(* IEC 61131-3 sources: Industry-PLC-LLM/data/PLCBEAD_repo/PLCBEAD_PLCEmbed-main/PLC-BEAD/Source/OpenPLCv2 (part 10) *)

(* ---- TN_SEND_ROWS.ST ---- *)
TYPE
  oscat_IP_FIFO128_DATA  : ARRAY [1..128] OF BYTE;
  oscat_Mailbox  : ARRAY [1..16] OF BYTE;

  oscat_IP_FIFO_DATA :
  STRUCT
    X       : oscat_IP_FIFO128_DATA; (* IP_ID FIFO Speicher          *)
    Y       : oscat_IP_FIFO128_DATA; (* IP_ID Z�hler                 *)
    ID      : BYTE;                  (* h�chste vergabene id         *)
    MAX_ID  : BYTE;                  (* maximal Anmeldungen pro ID   *)
    INIT    : BOOL;                  (* Initialisierung durchgef�hrt *)
    EMPTY   : BOOL;                  (* FIFO leer                    *)
    FULL    : BOOL;                  (* FIFO voll                    *)
    TOP     : INT;                   (* maximale anzahl in FIFO      *)
    NW      : INT;                   (* Schreibzeiger                *)
    NR      : INT;                   (* Lesezeiger                   *)
  END_STRUCT;

  oscat_IP_C:
  STRUCT
    C_MODE:			BYTE;          		(*W Mode: TCP/UCP AKTIV/PASSIV                               *)
    C_PORT:         WORD;          		(*W Portnummer                                               *)
    C_IP:           DWORD;         		(*W IP-Adresse gepackt wwxxyyzz = www.xxx.yyy.zzz            *)
    C_STATE:        BYTE;          		(*R Verbindungsstatus ON/OFF + Flanke ON/OFF                 *)
    C_ENABLE:       BOOL;          		(*W Freigabe f�r Connect                                     *)
    R_OBSERVE:      BOOL;          		(*W Empfang ueberwachen                                      *)
    TIME_RESET:     BOOL;          		(*W Alle Timer ruecksetzen                                   *)
    ERROR:          DWORD;         		(*R vvwwxxyy (vv = CON_ERROR, ww = SEN_ERROR, xx = REC_ERROR *)
    FIFO:           oscat_IP_FIFO_DATA; (*I IP FIFO Struktur                                         *)
    MAILBOX:		oscat_Mailbox;		(*I Mailbox: Datenbereich f�r Bausteindatenaustausch         *)
    END_STRUCT;
END_TYPE

TYPE

  oscat_NW_BUF_LONG  : ARRAY [0..4095] OF BYTE;

  oscat_NETWORK_BUFFER :
  STRUCT
    SIZE   : UINT;
    BUFFER : oscat_NW_BUF_LONG;
  END_STRUCT;

END_TYPE

TYPE

  bya_TN_CHAR:       	ARRAY [0..1919] OF BYTE;
  bya_TN_BACKUP:     	ARRAY [0..1919] OF BYTE;
  bya_TN_COLOR:      	ARRAY [0..1919] OF BYTE;
  bya_TN_Line_Update:	ARRAY [0..23]   OF BOOL;

  us_TN_SCREEN :
  STRUCT
    bya_CHAR:			bya_TN_CHAR;
    bya_COLOR:			bya_TN_COLOR;
    bya_BACKUP:			bya_TN_BACKUP;
    bya_Line_Update:	bya_TN_Line_Update;

    by_Input_Exten_Code:    BYTE;
    by_Input_ASCII_Code:    BYTE;
    bo_Input_ASCII_IsNum:   BOOL;
    in_Page_Number:        	INT;                (* aktive Seiten-Nr.              *)
    in_Cursor_X:           	INT;                (* Cursor X-Position              *)
    in_Cursor_Y:           	INT;                (* Cursor Y-Position              *)
    in_EOS_Offset:         	INT;                (* End of String Offset           *)
    by_Clear_Screen_Attr:  	BYTE;               (* Clear-Screen Attr              *)
    bo_Clear_Screen:       	BOOL;               (* Clear-Screen ausl�sen          *)
    bo_Modal_Dialog:       	BOOL;               (* Modaler Dialog ist aktiv       *)
    bo_Menue_Bar_Dialog:   	BOOL;               (* Menue Dialog ist aktiv         *)

  END_STRUCT;
END_TYPE

FUNCTION INT_TO_BCDC:BYTE

	VAR_INPUT
		IN :	INT;
	END_VAR

	INT_TO_BCDC := SHL(INT_TO_BYTE(IN / INT#10),4) OR INT_TO_BYTE(in MOD INT#10);

END_FUNCTION

FUNCTION_BLOCK TN_SEND_ROWS_Block

  VAR_IN_OUT
    IP_C :	oscat_IP_C;
    S_BUF :	oscat_NETWORK_BUFFER;
    Xus_TN_SCREEN :	us_TN_SCREEN;
  END_VAR

  VAR_INPUT
    S_BUF_SIZE :	INT;
  END_VAR

  VAR
    in_Line_Count :	INT;
    in_Col_Count :	INT;
    in_Last_Row_Index :	INT;
    bo_Break_Loop :	BOOL;
    in_Row_Count :	INT;
    in_Offset :	INT;
    in_Write_Index :	INT;
    in_Write_Index_Backup :	INT;
    by_Cur_Color :	BYTE;
    by_last_Color :	BYTE;
    in_Write_Stop :	INT;
  END_VAR

  IF (IP_C.C_STATE < BYTE#127 OR S_BUF.SIZE > UINT#0) THEN
    RETURN;
  END_IF;

  in_Write_Index := UINT_TO_INT(S_BUF.SIZE) - 1;

  in_Write_Index_Backup := in_Write_Index;

  IF (IP_C.C_STATE = BYTE#254) OR (Xus_TN_SCREEN.bo_Clear_Screen) THEN

    Xus_TN_SCREEN.bo_Clear_Screen := FALSE;

    FOR in_Line_Count := INT#00 TO INT#23 DO
      Xus_TN_SCREEN.bya_Line_Update[in_Line_Count] := TRUE;
    END_FOR;

    in_Write_Index := in_Write_Index + INT#1;
    S_BUF.BUFFER[in_Write_Index] := BYTE#16#1B;
    in_Write_Index := in_Write_Index + INT#1;
    S_BUF.BUFFER[in_Write_Index] := BYTE#16#5B;
    in_Write_Index := in_Write_Index + INT#1;
    S_BUF.BUFFER[in_Write_Index] := BYTE#16#30;
    in_Write_Index := in_Write_Index + INT#1;
    S_BUF.BUFFER[in_Write_Index] := BYTE#16#3B;
    in_Write_Index := in_Write_Index + INT#1;
    S_BUF.BUFFER[in_Write_Index] := BYTE#16#33;

    in_Write_Index := in_Write_Index + INT#1;
    S_BUF.BUFFER[in_Write_Index] := (SHR(Xus_TN_SCREEN.by_Clear_Screen_Attr,4) OR BYTE#16#30);

    in_Write_Index := in_Write_Index + INT#1;
    S_BUF.BUFFER[in_Write_Index] := BYTE#16#3B;
    in_Write_Index := in_Write_Index + INT#1;
    S_BUF.BUFFER[in_Write_Index] := BYTE#16#34;

    in_Write_Index := in_Write_Index + INT#1;
    S_BUF.BUFFER[in_Write_Index] := ((Xus_TN_SCREEN.by_Clear_Screen_Attr AND BYTE#16#07) OR BYTE#16#30);

    in_Write_Index := in_Write_Index + INT#1;
    S_BUF.BUFFER[in_Write_Index] := BYTE#16#6D;

    in_Write_Index := in_Write_Index + INT#1;
    S_BUF.BUFFER[in_Write_Index] := BYTE#16#1B;
    in_Write_Index := in_Write_Index + INT#1;
    S_BUF.BUFFER[in_Write_Index] := BYTE#16#5B;
    in_Write_Index := in_Write_Index + INT#1;
    S_BUF.BUFFER[in_Write_Index] := BYTE#16#32;
    in_Write_Index := in_Write_Index + INT#1;
    S_BUF.BUFFER[in_Write_Index] := BYTE#16#4A;

    in_Write_Index := in_Write_Index + INT#1;
    S_BUF.BUFFER[in_Write_Index] := BYTE#16#1B;
    in_Write_Index := in_Write_Index + INT#1;
    S_BUF.BUFFER[in_Write_Index] := BYTE#16#5B;
    in_Write_Index := in_Write_Index + INT#1;
    S_BUF.BUFFER[in_Write_Index] := BYTE#16#3F;
    in_Write_Index := in_Write_Index + INT#1;
    S_BUF.BUFFER[in_Write_Index] := BYTE#16#37;
    in_Write_Index := in_Write_Index + INT#1;
    S_BUF.BUFFER[in_Write_Index] := BYTE#16#6C;

  END_IF;

  in_Last_Row_Index := INT#0;
  bo_Break_Loop := FALSE;
  in_Write_Stop := S_BUF_SIZE-20;

  FOR in_Line_Count := 0 TO 23 DO

    in_Offset := in_Row_Count * INT#80;

    IF (Xus_TN_SCREEN.bya_Line_Update[in_Row_Count] = TRUE) THEN

      in_Write_Index := in_Write_Index + INT#1;
      S_BUF.BUFFER[in_Write_Index] := BYTE#16#1B;
      in_Write_Index := in_Write_Index + INT#1;
      S_BUF.BUFFER[in_Write_Index] := BYTE#16#5B;

      in_Write_Index := in_Write_Index + INT#1;
      S_BUF.BUFFER[in_Write_Index] :=
        SHR(INT_TO_BCDC(in_Row_Count + INT#1),INT#4) OR BYTE#16#30;

      in_Write_Index := in_Write_Index + INT#1;
      S_BUF.BUFFER[in_Write_Index] :=
        (INT_TO_BCDC(in_Row_Count + INT#1) AND BYTE#16#0F) OR BYTE#16#30;

      in_Write_Index := in_Write_Index + INT#1;
      S_BUF.BUFFER[in_Write_Index] := BYTE#16#3B;
      in_Write_Index := in_Write_Index + INT#1;
      S_BUF.BUFFER[in_Write_Index] := BYTE#16#31;
      in_Write_Index := in_Write_Index + INT#1;
      S_BUF.BUFFER[in_Write_Index] := BYTE#16#48;

      FOR in_Col_Count := 0 TO 79 DO

        by_Cur_Color := Xus_TN_SCREEN.bya_COLOR[in_Offset];
        IF (by_Cur_Color <> by_last_Color) OR (in_Col_Count = INT#00) THEN

          in_Write_Index := in_Write_Index + INT#1;
          S_BUF.BUFFER[in_Write_Index] := BYTE#16#1B;

          in_Write_Index := in_Write_Index + INT#1;
          S_BUF.BUFFER[in_Write_Index] := BYTE#16#5B;

          IF  (((by_Cur_Color AND BYTE#2#10001000) XOR (by_last_Color AND BYTE#2#10001000)) <> BYTE#00) OR (in_Col_Count = 0) THEN

            in_Write_Index := in_Write_Index + INT#1;
            S_BUF.BUFFER[in_Write_Index] := BYTE#16#30;
            in_Write_Index := in_Write_Index + INT#1;
            S_BUF.BUFFER[in_Write_Index] := BYTE#16#3B;

            IF (by_Cur_Color AND BYTE#2#00001000) = BYTE#2#00000000 THEN

              in_Write_Index := in_Write_Index + INT#1;
              S_BUF.BUFFER[in_Write_Index] := BYTE#16#31;
              in_Write_Index := in_Write_Index + INT#1;
              S_BUF.BUFFER[in_Write_Index] := BYTE#16#3B;

            END_IF;

            IF (by_Cur_Color AND BYTE#2#10000000) = BYTE#2#10000000 THEN

              in_Write_Index := in_Write_Index + INT#1;
              S_BUF.BUFFER[in_Write_Index] := BYTE#16#35;
              in_Write_Index := in_Write_Index + INT#1;
              S_BUF.BUFFER[in_Write_Index] := BYTE#16#3B;

            END_IF;

          END_IF;

          in_Write_Index := in_Write_Index + INT#1;
          S_BUF.BUFFER[in_Write_Index] := BYTE#16#33;

          in_Write_Index := in_Write_Index + INT#1;
          S_BUF.BUFFER[in_Write_Index] := ((SHR(by_Cur_Color,4) AND BYTE#2#00000111) OR BYTE#16#30);

          in_Write_Index := in_Write_Index + INT#1;
          S_BUF.BUFFER[in_Write_Index] := BYTE#16#3B;

          in_Write_Index := in_Write_Index + INT#1;
          S_BUF.BUFFER[in_Write_Index] := BYTE#16#34;

          in_Write_Index := in_Write_Index + INT#1;
          S_BUF.BUFFER[in_Write_Index] := ((by_Cur_Color AND BYTE#2#00000111) OR BYTE#16#30);

          in_Write_Index := in_Write_Index + INT#1;
          S_BUF.BUFFER[in_Write_Index] := BYTE#16#6D;

          by_last_Color := by_Cur_Color;

        END_IF;

        IF (in_Write_Index > in_Write_Stop) THEN

          bo_Break_Loop := TRUE;
          EXIT;

        END_IF;

        in_Write_Index := in_Write_Index + INT#1;
        S_BUF.BUFFER[in_Write_Index] := Xus_TN_SCREEN.bya_CHAR[in_Offset];

        in_Offset := in_Offset + INT#01;
      END_FOR;

      IF (bo_Break_Loop = TRUE) THEN

        in_Write_Index := in_Last_Row_Index;

        EXIT;
      END_IF;

      in_Last_Row_Index := in_Write_Index;
      Xus_TN_SCREEN.bya_Line_Update[in_Row_Count] := FALSE;

    END_IF;

    in_Row_Count := in_Row_Count + INT#01;

    IF (in_Row_Count > INT#23) THEN
      in_Row_Count := INT#00;
    END_IF;

  END_FOR;

  IF (bo_Break_Loop = FALSE) THEN

    in_Row_Count := INT#00;

  END_IF;

  IF (in_Write_Index <> in_Write_Index_Backup) THEN

    in_Write_Index := in_Write_Index + INT#1;
    S_BUF.BUFFER[in_Write_Index] := BYTE#16#1B;
    in_Write_Index := in_Write_Index + INT#1;
    S_BUF.BUFFER[in_Write_Index] := BYTE#16#5B;

    in_Write_Index := in_Write_Index + INT#1;
    S_BUF.BUFFER[in_Write_Index] := SHR(INT_TO_BCDC(Xus_TN_SCREEN.in_Cursor_Y + 1),INT#4) OR BYTE#16#30;

    in_Write_Index := in_Write_Index + INT#1;
    S_BUF.BUFFER[in_Write_Index] := (INT_TO_BCDC(Xus_TN_SCREEN.in_Cursor_Y + 1) AND BYTE#16#0F) OR BYTE#16#30;

    in_Write_Index := in_Write_Index + INT#1;
    S_BUF.BUFFER[in_Write_Index] := BYTE#16#3B;

    in_Write_Index := in_Write_Index + INT#1;
    S_BUF.BUFFER[in_Write_Index] := SHR(INT_TO_BCDC(Xus_TN_SCREEN.in_Cursor_X + 1),INT#4) OR BYTE#16#30;

    in_Write_Index := in_Write_Index + INT#1;
    S_BUF.BUFFER[in_Write_Index] := (INT_TO_BCDC(Xus_TN_SCREEN.in_Cursor_X + 1) AND BYTE#16#0F) OR BYTE#16#30;

    in_Write_Index := in_Write_Index + INT#1;
    S_BUF.BUFFER[in_Write_Index] := BYTE#16#48;

  END_IF;

  S_BUF.SIZE := INT_TO_UINT(in_Write_Index + 1);

END_FUNCTION_BLOCK

PROGRAM program0
	VAR
		IP_C :	oscat_IP_C;
    S_BUF :	oscat_NETWORK_BUFFER;
    Xus_TN_SCREEN :	us_TN_SCREEN;
    S_BUF_SIZE :	INT;

		func_block : TN_SEND_ROWS_Block;
	END_VAR
	func_block.IP_C := IP_C;
  func_block.S_BUF := S_BUF;
  func_block.Xus_TN_SCREEN := Xus_TN_SCREEN;
  func_block.S_BUF_SIZE := S_BUF_SIZE;

	func_block();
	IP_C  := func_block.IP_C;
  S_BUF  := func_block.S_BUF;
  Xus_TN_SCREEN  := func_block.Xus_TN_SCREEN;
END_PROGRAM

CONFIGURATION Config0
	RESOURCE Res0 ON PLC
		TASK task0(INTERVAL := T#20ms,PRIORITY := 0);
		PROGRAM instance0 WITH task0 : program0;
	END_RESOURCE
END_CONFIGURATION

(* ---- TO_UML.ST ---- *)
FUNCTION _BYTE_TO_INT:INT
	VAR_INPUT
		IN :	BYTE;
	END_VAR

	_BYTE_TO_INT := USINT_TO_INT(BYTE_TO_USINT(IN));
END_FUNCTION

FUNCTION_BLOCK TO_UML_Block

	VAR_INPUT
		IN :	BYTE;
	END_VAR

	VAR_OUTPUT
		TO_UML :	STRING;
	END_VAR

	CASE _BYTE_TO_INT(in) OF
		196:
			TO_UML := 'Ae';
		214:
			TO_UML := 'Oe';
		220:
			TO_UML := 'Ue';
		223:
			TO_UML := 'ss';
		228:
			TO_UML := 'ae';
		246:
			TO_UML := 'oe';
		252:
			TO_UML := 'ue';
	ELSE
		TO_UML := BYTE_TO_STRING(IN);
	END_CASE;

END_FUNCTION_BLOCK

PROGRAM program0
  VAR
	IN :	BYTE;
	TO_UML :	STRING;
	func_block : TO_UML_Block;
  END_VAR
	func_block.IN  := IN;
	func_block();
	TO_UML := func_block.TO_UML;

END_PROGRAM

CONFIGURATION Config0
	RESOURCE Res0 ON PLC
		TASK task0(INTERVAL := T#20ms,PRIORITY := 0);
		PROGRAM instance0 WITH task0 : program0;
	END_RESOURCE
END_CONFIGURATION

(* ---- TOD_TO_STRING.ST ---- *)
FUNCTION HOUR:INT
	VAR_INPUT
		ITOD :	UDINT;
	END_VAR
	hour := UDINT_TO_INT(itod / UDINT#3600000);
END_FUNCTION

FUNCTION MINUTE:INT

	VAR_INPUT
		ITOD :	UDINT;
	END_VAR

	minute := UDINT_TO_INT((itod / UDINT#60000) - ((itod / UDINT#3600000) * UDINT#60));

END_FUNCTION

FUNCTION_BLOCK TOD_TO_STRING_Block
	VAR_INPUT
		ITOD :	UDINT;
	END_VAR

	VAR_OUTPUT
		TOD_STRING :	STRING;
	END_VAR

	VAR
		st_tmp1 :	STRING;
		st_tmp2 :	STRING;
		cur_hours :	INT;
	END_VAR

	cur_hours := hour(ITOD);
	IF cur_hours = 0 THEN
	st_tmp2 := '%01dh';
	ELSE
	st_tmp2 := '%dh';
	END_IF;

	st_tmp1 := CONCAT(INT_TO_STRING(cur_hours),INT_TO_STRING(minute(ITOD)));
	TOD_STRING := CONCAT(st_tmp1,UDINT_TO_STRING(ITOD MOD UDINT#60000 / UDINT#1000));
END_FUNCTION_BLOCK

PROGRAM program0
  VAR
    LocalVar0 : UDINT;
	LocalOUT  : STRING;
	func_block : TOD_TO_STRING_Block;
  END_VAR
	func_block.ITOD  := LocalVar0;
	func_block();
	LocalOUT := func_block.TOD_STRING;
END_PROGRAM

CONFIGURATION Config0
  RESOURCE Res0 ON PLC
    TASK task0(INTERVAL := T#20ms,PRIORITY := 0);
    PROGRAM instance0 WITH task0 : program0;
  END_RESOURCE
END_CONFIGURATION

(* ---- TOF_1.ST ---- *)
FUNCTION UDINT_TO_TIME2:TIME

	VAR_INPUT
		IN :	UDINT;
	END_VAR

	UDINT_TO_TIME2 := DINT_TO_TIME(UDINT_TO_DINT(IN));

END_FUNCTION

FUNCTION_BLOCK T_PLC_MS_block
	VAR_OUTPUT
		T_PLC_MS :	UDINT;
	END_VAR

	VAR_EXTERNAL
		PLC_TICKS_PER_SEC :	INT;
		PLC_SYS_TICK_CNT :	DINT;
	END_VAR

	VAR
		debug :	BOOL;(*Debug-Mode ON / OFF*)
		N :	INT;(*Debug-Faktor*)
		Offset :	UDINT;(*Debug-Offset*)
		temp :	DWORD := DWORD#1;(*Debug-Offset*)
		mode :	BOOL;(*modus*)
		faktor :	UDINT;(*Systemtakt-Faktor*)
		init :	BOOL;
		v_plc_ticks_per_sec :	UDINT;
		base :	UDINT := UDINT#1000;
	END_VAR

	IF init = FALSE THEN
		v_plc_ticks_per_sec := INT_TO_UDINT(PLC_TICKS_PER_SEC);
		IF v_plc_ticks_per_sec = UDINT#1024 THEN
			faktor := UDINT#1;
			mode := FALSE;
		ELSIF v_plc_ticks_per_sec > UDINT#0 THEN
			IF v_plc_ticks_per_sec <= base THEN
				faktor := base / v_plc_ticks_per_sec;
				mode := FALSE;
			ELSE
				faktor := v_plc_ticks_per_sec / base;
				mode := TRUE;
			END_IF;
		ELSE
			faktor := UDINT#1;
		END_IF;
		init := TRUE;
	END_IF;

	IF mode THEN
		T_PLC_MS := DINT_TO_UDINT(PLC_SYS_TICK_CNT) / faktor;
	ELSE
		T_PLC_MS := DINT_TO_UDINT(PLC_SYS_TICK_CNT) * faktor;
	END_IF;

	IF debug THEN
		T_PLC_MS := (DWORD_TO_UDINT(SHL(UDINT_TO_DWORD(T_PLC_MS),N) OR SHL(temp,N)) - UDINT#1) + Offset;
	END_IF;

END_FUNCTION_BLOCK

FUNCTION_BLOCK TOF_1

	VAR_INPUT
		IN :	BOOL;
		PT :	TIME;
		RST :	BOOL;
	END_VAR

	VAR_OUTPUT
		Q :	BOOL;
	END_VAR

	VAR
		start :	TIME;
		tx :	TIME;
		T_PLC_MS :	T_PLC_MS_block;
	END_VAR

	T_PLC_MS();
	tx:= UDINT_TO_TIME(T_PLC_MS.T_PLC_MS);

	IF RST THEN
		Q := FALSE;
	ELSIF IN THEN
		Q := TRUE;
		start := tx;
	ELSIF tx - start >= PT THEN
		Q := FALSE;
	END_IF;

END_FUNCTION_BLOCK

PROGRAM program0
  VAR
	IN :	BOOL;
	PT :	TIME;
	RST :	BOOL;
	Q :	BOOL;
	func_block : TOF_1;
  END_VAR
	func_block.IN  :=IN;
	func_block.PT  :=PT;
	func_block.RST  :=RST;
	func_block();
	Q := func_block.Q;
END_PROGRAM

CONFIGURATION Config0
	VAR_GLOBAL
		PLC_TICKS_PER_SEC :	INT;
		PLC_SYS_TICK_CNT :	DINT;
	END_VAR
	RESOURCE Res0 ON PLC
		TASK task0(INTERVAL := T#20ms,PRIORITY := 0);
		PROGRAM instance0 WITH task0 : program0;
	END_RESOURCE
END_CONFIGURATION

(* ---- TOGGLE.ST ---- *)
FUNCTION_BLOCK TOGGLE

	VAR_INPUT
		CLK :	BOOL;
		RST :	BOOL;
	END_VAR

	VAR_OUTPUT
		Q :	BOOL;
	END_VAR

	VAR
		edge :	BOOL;
	END_VAR

	IF rst THEN
		Q := FALSE;
	ELSIF clk AND NOT edge THEN
		Q := NOT Q;
	END_IF;
	edge := clk;

END_FUNCTION_BLOCK

PROGRAM program0
  VAR
	CLK :	BOOL;
	RST :	BOOL;
	Q :	BOOL;
	func_block : TOGGLE;
  END_VAR
	func_block.CLK  :=CLK;
	func_block.RST  :=RST;
	func_block();
	Q := func_block.Q;

END_PROGRAM

CONFIGURATION Config0
	RESOURCE Res0 ON PLC
		TASK task0(INTERVAL := T#20ms,PRIORITY := 0);
		PROGRAM instance0 WITH task0 : program0;
	END_RESOURCE
END_CONFIGURATION

(* ---- TONOF.ST ---- *)
FUNCTION_BLOCK TONOF

	VAR_INPUT
		IN :	BOOL;
		T_ON :	TIME;
		T_OFF :	TIME;
	END_VAR

	VAR_OUTPUT
		Q :	BOOL;
	END_VAR

	VAR
		X :	TON;
		old :	BOOL;
		mode :	BOOL;
	END_VAR

	IF IN XOR old THEN
	X(IN := FALSE, PT := SEL_TIME(IN,T_OFF,T_ON));
	mode := IN;
	old := IN;
	END_IF;
	X(IN := TRUE);
	IF X.Q THEN Q := mode;END_IF;

END_FUNCTION_BLOCK

PROGRAM program0
  VAR
	IN :	BOOL;
	T_ON :	TIME;
	T_OFF :	TIME;
	Q :	BOOL;
	func_block : TONOF;
  END_VAR
	func_block.IN  :=IN ;
	func_block.T_ON  :=T_ON ;
	func_block.T_OFF  :=T_OFF ;
	func_block();
	Q := func_block.Q;

END_PROGRAM

CONFIGURATION Config0
	RESOURCE Res0 ON PLC
		TASK task0(INTERVAL := T#20ms,PRIORITY := 0);
		PROGRAM instance0 WITH task0 : program0;
	END_RESOURCE
END_CONFIGURATION

(* ---- TP_1.ST ---- *)
FUNCTION UDINT_TO_TIME2:TIME

	VAR_INPUT
		IN :	UDINT;
	END_VAR

	UDINT_TO_TIME2 := DINT_TO_TIME(UDINT_TO_DINT(IN));

END_FUNCTION

FUNCTION_BLOCK T_PLC_MS_block
	VAR_OUTPUT
		T_PLC_MS :	UDINT;
	END_VAR

	VAR_EXTERNAL
		PLC_TICKS_PER_SEC :	INT;
		PLC_SYS_TICK_CNT :	DINT;
	END_VAR

	VAR
		debug :	BOOL;(*Debug-Mode ON / OFF*)
		N :	INT;(*Debug-Faktor*)
		Offset :	UDINT;(*Debug-Offset*)
		temp :	DWORD := DWORD#1;(*Debug-Offset*)
		mode :	BOOL;(*modus*)
		faktor :	UDINT;(*Systemtakt-Faktor*)
		init :	BOOL;
		v_plc_ticks_per_sec :	UDINT;
		base :	UDINT := UDINT#1000;
	END_VAR

	IF init = FALSE THEN
		v_plc_ticks_per_sec := INT_TO_UDINT(PLC_TICKS_PER_SEC);
		IF v_plc_ticks_per_sec = UDINT#1024 THEN
			faktor := UDINT#1;
			mode := FALSE;
		ELSIF v_plc_ticks_per_sec > UDINT#0 THEN
			IF v_plc_ticks_per_sec <= base THEN
				faktor := base / v_plc_ticks_per_sec;
				mode := FALSE;
			ELSE
				faktor := v_plc_ticks_per_sec / base;
				mode := TRUE;
			END_IF;
		ELSE
			faktor := UDINT#1;
		END_IF;
		init := TRUE;
	END_IF;

	IF mode THEN
		T_PLC_MS := DINT_TO_UDINT(PLC_SYS_TICK_CNT) / faktor;
	ELSE
		T_PLC_MS := DINT_TO_UDINT(PLC_SYS_TICK_CNT) * faktor;
	END_IF;

	IF debug THEN
		T_PLC_MS := (DWORD_TO_UDINT(SHL(UDINT_TO_DWORD(T_PLC_MS),N) OR SHL(temp,N)) - UDINT#1) + Offset;
	END_IF;

END_FUNCTION_BLOCK

FUNCTION_BLOCK TP_1

	VAR_INPUT
		IN :	BOOL;
		PT :	TIME;
		RST :	BOOL;
	END_VAR

	VAR_OUTPUT
		Q :	BOOL;
	END_VAR

	VAR
		tx :	TIME;
		start :	TIME;
		ix :	BOOL;
		T_PLC_MS :	T_PLC_MS_block;
	END_VAR

	T_PLC_MS();
	tx := UDINT_TO_TIME(T_PLC_MS.T_PLC_MS);

	IF RST THEN
		Q := FALSE;
	ELSIF IN AND NOT ix THEN
		Q := TRUE;
		start := tx;
	ELSIF tx - start >= PT THEN
		Q := FALSE;
	END_IF;

	ix:= IN;

END_FUNCTION_BLOCK

PROGRAM program0
  VAR
	IN :	BOOL;
	PT :	TIME;
	RST :	BOOL;
	Q :	BOOL;
	func_block : TP_1;
  END_VAR
	func_block.IN  :=IN;
	func_block.PT  :=PT;
	func_block.RST  :=RST;
	func_block();
	Q := func_block.Q;
END_PROGRAM

CONFIGURATION Config0
	VAR_GLOBAL
		PLC_TICKS_PER_SEC :	INT;
		PLC_SYS_TICK_CNT :	DINT;
	END_VAR
	RESOURCE Res0 ON PLC
		TASK task0(INTERVAL := T#20ms,PRIORITY := 0);
		PROGRAM instance0 WITH task0 : program0;
	END_RESOURCE
END_CONFIGURATION

(* ---- TP_1D.ST ---- *)
FUNCTION UDINT_TO_TIME2:TIME

	VAR_INPUT
		IN :	UDINT;
	END_VAR

	UDINT_TO_TIME2 := DINT_TO_TIME(UDINT_TO_DINT(IN));

END_FUNCTION

FUNCTION_BLOCK T_PLC_MS_block
	VAR_OUTPUT
		T_PLC_MS :	UDINT;
	END_VAR

	VAR_EXTERNAL
		PLC_TICKS_PER_SEC :	INT;
		PLC_SYS_TICK_CNT :	DINT;
	END_VAR

	VAR
		debug :	BOOL;(*Debug-Mode ON / OFF*)
		N :	INT;(*Debug-Faktor*)
		Offset :	UDINT;(*Debug-Offset*)
		temp :	DWORD := DWORD#1;(*Debug-Offset*)
		mode :	BOOL;(*modus*)
		faktor :	UDINT;(*Systemtakt-Faktor*)
		init :	BOOL;
		v_plc_ticks_per_sec :	UDINT;
		base :	UDINT := UDINT#1000;
	END_VAR

	IF init = FALSE THEN
		v_plc_ticks_per_sec := INT_TO_UDINT(PLC_TICKS_PER_SEC);
		IF v_plc_ticks_per_sec = UDINT#1024 THEN
			faktor := UDINT#1;
			mode := FALSE;
		ELSIF v_plc_ticks_per_sec > UDINT#0 THEN
			IF v_plc_ticks_per_sec <= base THEN
				faktor := base / v_plc_ticks_per_sec;
				mode := FALSE;
			ELSE
				faktor := v_plc_ticks_per_sec / base;
				mode := TRUE;
			END_IF;
		ELSE
			faktor := UDINT#1;
		END_IF;
		init := TRUE;
	END_IF;

	IF mode THEN
		T_PLC_MS := DINT_TO_UDINT(PLC_SYS_TICK_CNT) / faktor;
	ELSE
		T_PLC_MS := DINT_TO_UDINT(PLC_SYS_TICK_CNT) * faktor;
	END_IF;

	IF debug THEN
		T_PLC_MS := (DWORD_TO_UDINT(SHL(UDINT_TO_DWORD(T_PLC_MS),N) OR SHL(temp,N)) - UDINT#1) + Offset;
	END_IF;

END_FUNCTION_BLOCK

FUNCTION_BLOCK TP_1D
	VAR_INPUT
		IN :	BOOL;
		PT1 :	TIME;
		PTD :	TIME;
		RST :	BOOL;
	END_VAR

	VAR_OUTPUT
		Q :	BOOL;
		W :	BOOL;
	END_VAR

	VAR
		tx :	TIME;
		start :	TIME;
		ix :	BOOL;
		T_PLC_MS :	T_PLC_MS_block;
	END_VAR

	T_PLC_MS();
	tx := UDINT_TO_TIME(T_PLC_MS.T_PLC_MS);

	IF RST THEN
		Q := FALSE;
		rst := FALSE;
		W := FALSE;
	ELSIF W THEN
		IF tx - start >= PTD THEN
			W := FALSE;
		END_IF;
	ELSIF IN AND NOT ix THEN
		Q := TRUE;
		start := tx;
		in := FALSE;
	ELSIF tx - start >= PT1 THEN
		Q := FALSE;
		W := TRUE;
		start := tx;
	END_IF;

	ix := IN;

END_FUNCTION_BLOCK

PROGRAM program0
  VAR
	IN :	BOOL;
	PT1 :	TIME;
	PTD :	TIME;
	RST :	BOOL;
	Q :	BOOL;
	W :	BOOL;
	func_block : TP_1D;
  END_VAR
	func_block.IN  :=IN;
	func_block.PT1  :=PT1;
	func_block.PTD  :=PTD;
	func_block.RST  :=RST;
	func_block();
	Q := func_block.Q;
	W := func_block.W;
END_PROGRAM

CONFIGURATION Config0
	VAR_GLOBAL
		PLC_TICKS_PER_SEC :	INT;
		PLC_SYS_TICK_CNT :	DINT;
	END_VAR
	RESOURCE Res0 ON PLC
		TASK task0(INTERVAL := T#20ms,PRIORITY := 0);
		PROGRAM instance0 WITH task0 : program0;
	END_RESOURCE
END_CONFIGURATION

(* ---- TP_X.ST ---- *)
FUNCTION UDINT_TO_TIME2:TIME

	VAR_INPUT
		IN :	UDINT;
	END_VAR

	UDINT_TO_TIME2 := DINT_TO_TIME(UDINT_TO_DINT(IN));

END_FUNCTION

FUNCTION_BLOCK T_PLC_MS_block
	VAR_OUTPUT
		T_PLC_MS :	UDINT;
	END_VAR

	VAR_EXTERNAL
		PLC_TICKS_PER_SEC :	INT;
		PLC_SYS_TICK_CNT :	DINT;
	END_VAR

	VAR
		debug :	BOOL;(*Debug-Mode ON / OFF*)
		N :	INT;(*Debug-Faktor*)
		Offset :	UDINT;(*Debug-Offset*)
		temp :	DWORD := DWORD#1;(*Debug-Offset*)
		mode :	BOOL;(*modus*)
		faktor :	UDINT;(*Systemtakt-Faktor*)
		init :	BOOL;
		v_plc_ticks_per_sec :	UDINT;
		base :	UDINT := UDINT#1000;
	END_VAR

	IF init = FALSE THEN
		v_plc_ticks_per_sec := INT_TO_UDINT(PLC_TICKS_PER_SEC);
		IF v_plc_ticks_per_sec = UDINT#1024 THEN
			faktor := UDINT#1;
			mode := FALSE;
		ELSIF v_plc_ticks_per_sec > UDINT#0 THEN
			IF v_plc_ticks_per_sec <= base THEN
				faktor := base / v_plc_ticks_per_sec;
				mode := FALSE;
			ELSE
				faktor := v_plc_ticks_per_sec / base;
				mode := TRUE;
			END_IF;
		ELSE
			faktor := UDINT#1;
		END_IF;
		init := TRUE;
	END_IF;

	IF mode THEN
		T_PLC_MS := DINT_TO_UDINT(PLC_SYS_TICK_CNT) / faktor;
	ELSE
		T_PLC_MS := DINT_TO_UDINT(PLC_SYS_TICK_CNT) * faktor;
	END_IF;

	IF debug THEN
		T_PLC_MS := (DWORD_TO_UDINT(SHL(UDINT_TO_DWORD(T_PLC_MS),N) OR SHL(temp,N)) - UDINT#1) + Offset;
	END_IF;

END_FUNCTION_BLOCK

FUNCTION_BLOCK TP_X
	VAR_INPUT
		IN :	BOOL;
		PT :	TIME;
	END_VAR

	VAR_OUTPUT
		Q :	BOOL;
		ET :	TIME;
	END_VAR

	VAR
		edge :	BOOL;
		start :	TIME;
		tx :	TIME;
		T_PLC_MS :	T_PLC_MS_block;
	END_VAR

	T_PLC_MS();
	tx := UDINT_TO_TIME2(T_PLC_MS.T_PLC_MS);

	IF IN AND NOT edge THEN
		start := tx;
		Q := PT > t#0ms;
	ELSIF Q THEN
		ET := tx - start;
		IF ET >= PT THEN
			Q := FALSE;
			ET := t#0ms;
		END_IF;
	END_IF;
	edge := IN;

END_FUNCTION_BLOCK

PROGRAM program0
  VAR
	IN :	BOOL;
	PT :	TIME;
	Q :	BOOL;
	ET :	TIME;
	func_block : TP_X;
  END_VAR
	func_block.IN  :=IN;
	func_block.PT  :=PT ;
	func_block();
	Q := func_block.Q;
	ET := func_block.ET;
END_PROGRAM

CONFIGURATION Config0
	VAR_GLOBAL
		PLC_TICKS_PER_SEC :	INT;
		PLC_SYS_TICK_CNT :	DINT;
	END_VAR
	RESOURCE Res0 ON PLC
		TASK task0(INTERVAL := T#20ms,PRIORITY := 0);
		PROGRAM instance0 WITH task0 : program0;
	END_RESOURCE
END_CONFIGURATION

(* ---- TREND.ST ---- *)
FUNCTION_BLOCK TREND

	VAR_INPUT
		X :	REAL;
	END_VAR

	VAR_OUTPUT
		Q :	BOOL;
		TU :	BOOL;
		TD :	BOOL;
		D :	REAL;
	END_VAR

	VAR
		last_x :	REAL;
	END_VAR

	TU := X > last_X;
	TD := X < last_X;
	Q := TU OR TD;
	D := X - LAST_X;

	last_X := X;

END_FUNCTION_BLOCK

PROGRAM program0
  VAR
	X :	REAL;
	Q :	BOOL;
	TU :	BOOL;
	TD :	BOOL;
	D :	REAL;
	func_block : TREND;
  END_VAR
	func_block.X  :=X ;
	func_block();
	Q := func_block.Q;
	TU := func_block.TU;
	TD := func_block.TD;
	D := func_block.D;
END_PROGRAM

CONFIGURATION Config0
	RESOURCE Res0 ON PLC
		TASK task0(INTERVAL := T#20ms,PRIORITY := 0);
		PROGRAM instance0 WITH task0 : program0;
	END_RESOURCE
END_CONFIGURATION

(* ---- TREND_DW.ST ---- *)
FUNCTION_BLOCK TREND_DW
	VAR_INPUT
		X :	DWORD;
	END_VAR
	VAR_OUTPUT
		Q :	BOOL;
		TU :	BOOL;
		TD :	BOOL;
		D :	DWORD;
	END_VAR

	VAR
		LAST_X :	DWORD;
	END_VAR

	IF X > last_X THEN
		TU := TRUE;
		TD := FALSE;
		D := UDINT_TO_DWORD(DWORD_TO_UDINT(X) - DWORD_TO_UDINT(last_X));
		Q := TRUE;
	ELSIF X < last_X THEN
		TD := TRUE;
		TU := FALSE;
		D := UDINT_TO_DWORD(DWORD_TO_UDINT(last_X) - DWORD_TO_UDINT(X));
		Q := FALSE;
	ELSE
		TU := FALSE;
		TD := FALSE;
		D := DWORD#0;
	END_IF;
	last_X := X;
END_FUNCTION_BLOCK

PROGRAM program0
  VAR
	X :	DWORD;
	Q :	BOOL;
	TU :	BOOL;
	TD :	BOOL;
	D :	DWORD;
	func_block : TREND_DW;
  END_VAR
	func_block.X  :=X ;
	func_block();
	Q := func_block.Q;
	TU := func_block.TU;
	TD := func_block.TD;
	D := func_block.D;
END_PROGRAM

CONFIGURATION Config0
	RESOURCE Res0 ON PLC
		TASK task0(INTERVAL := T#20ms,PRIORITY := 0);
		PROGRAM instance0 WITH task0 : program0;
	END_RESOURCE
END_CONFIGURATION

(* ---- TRIM.ST ---- *)
FUNCTION_BLOCK TRIM

	VAR_INPUT
		STR :	STRING;
	END_VAR

	VAR_OUTPUT
		TRIM3 :	STRING;
	END_VAR

	VAR
		pos :	INT;
	END_VAR

	trim3 := str;
	REPEAT
		pos := FIND(trim3,' ');
		IF pos > 0 THEN trim3 := REPLACE(trim3,'',1,pos); END_IF;
	UNTIL pos = 0 END_REPEAT;

END_FUNCTION_BLOCK

PROGRAM program0
  VAR
	STR :	STRING;

	TRIM3 :	STRING;
	func_block : TRIM;
  END_VAR
	func_block.STR  :=STR ;
	func_block();
	TRIM3 := func_block.TRIM3;

END_PROGRAM

CONFIGURATION Config0
	RESOURCE Res0 ON PLC
		TASK task0(INTERVAL := T#20ms,PRIORITY := 0);
		PROGRAM instance0 WITH task0 : program0;
	END_RESOURCE
END_CONFIGURATION

(* ---- TRIM1.ST ---- *)
FUNCTION_BLOCK TRIM1

	VAR_INPUT
		STR :	STRING;
	END_VAR

	VAR_OUTPUT
		TRIM3 :	STRING;
	END_VAR

	VAR
		pos :	INT;
		st_temp :	STRING;
	END_VAR

	trim3 := str;
	REPEAT
		pos := FIND(trim3,'  ');
		IF pos > 0 THEN
		st_temp := trim3;
		trim3 := REPLACE(trim3,' ',2,pos);
		END_IF;
	UNTIL pos = 0 END_REPEAT;
	st_temp := LEFT(trim3,1);
	IF EQ_STRING(st_temp,' ') THEN trim3 := DELETE(trim3,1,1); END_IF;
	st_temp := RIGHT(trim3,1);
	IF EQ_STRING(st_temp,' ') THEN trim3 := DELETE(trim3,1,LEN(trim3)); END_IF;

END_FUNCTION_BLOCK

PROGRAM program0
  VAR
	STR :	STRING;

	TRIM3 :	STRING;
	func_block : TRIM1;
  END_VAR
	func_block.STR  :=STR ;
	func_block();
	TRIM3 := func_block.TRIM3;

END_PROGRAM

CONFIGURATION Config0
	RESOURCE Res0 ON PLC
		TASK task0(INTERVAL := T#20ms,PRIORITY := 0);
		PROGRAM instance0 WITH task0 : program0;
	END_RESOURCE
END_CONFIGURATION

(* ---- TUNE.ST ---- *)
FUNCTION_BLOCK T_PLC_MS_Block
	VAR_OUTPUT
		T_PLC_MS :	UDINT;
	END_VAR

	VAR_EXTERNAL
		PLC_TICKS_PER_SEC :	INT;
		PLC_SYS_TICK_CNT :	DINT;
	END_VAR

	VAR
		debug :	BOOL;(*Debug-Mode ON / OFF*)
		N :	INT;(*Debug-Faktor*)
		Offset :	UDINT;(*Debug-Offset*)
		temp :	DWORD := DWORD#1;(*Debug-Offset*)
		mode :	BOOL;(*modus*)
		faktor :	UDINT;(*Systemtakt-Faktor*)
		init :	BOOL;
		v_plc_ticks_per_sec :	UDINT;
		base :	UDINT := UDINT#1000;
	END_VAR

	IF init = FALSE THEN
		v_plc_ticks_per_sec := INT_TO_UDINT(PLC_TICKS_PER_SEC);
		IF v_plc_ticks_per_sec = UDINT#1024 THEN
			faktor := UDINT#1;
			mode := FALSE;
		ELSIF v_plc_ticks_per_sec > UDINT#0 THEN
			IF v_plc_ticks_per_sec <= base THEN
				faktor := base / v_plc_ticks_per_sec;
				mode := FALSE;
			ELSE
				faktor := v_plc_ticks_per_sec / base;
				mode := TRUE;
			END_IF;
		ELSE
			faktor := UDINT#1;
		END_IF;
		init := TRUE;
	END_IF;

	IF mode THEN
		T_PLC_MS := DINT_TO_UDINT(PLC_SYS_TICK_CNT) / faktor;
	ELSE
		T_PLC_MS := DINT_TO_UDINT(PLC_SYS_TICK_CNT) * faktor;
	END_IF;

	IF debug THEN
		T_PLC_MS := (DWORD_TO_UDINT(SHL(UDINT_TO_DWORD(T_PLC_MS),N) OR SHL(temp,N)) - UDINT#1) + Offset;
	END_IF;
END_FUNCTION_BLOCK

FUNCTION TIME_TO_UDINT2:UDINT
	VAR_INPUT
		X :	TIME;
	END_VAR

	TIME_TO_UDINT2 := DINT_TO_UDINT(TIME_TO_DINT(X));
END_FUNCTION

FUNCTION_BLOCK TUNE_Block

	VAR_INPUT
		SET :	BOOL;
		SU :	BOOL;
		SD :	BOOL;
		RST :	BOOL;
		SS :	REAL := 0.1;
		LIMIT_L :	REAL;
		LIMIT_H :	REAL := 100.0;
		RST_VAL :	REAL;
		SET_VAL :	REAL := 100.0;
		T1 :	TIME := T#500ms;
		T2 :	TIME := T#2s;
		S1 :	REAL := 2.0;
		S2 :	REAL := 10.0;
	END_VAR

	VAR_OUTPUT
		Y :	REAL;
	END_VAR

	VAR
		tx :	UDINT;
		start :	UDINT;
		start2 :	UDINT;
		state :	INT;
		in :	BOOL;
		step2 :	REAL;
		speed :	REAL;
		Y_start :	REAL;
		Y_start2 :	REAL;
		T_PLC_MS :	T_PLC_MS_Block;
	END_VAR

	T_PLC_MS();
	tx:= T_PLC_MS.T_PLC_MS;

	IF rst THEN
		Y := RST_val;
		state := 0;
	ELSIF set THEN
		Y := SET_val;
		state := 0;
	ELSIF state > 0 THEN
		IF state = 1 THEN
			in := su;
		ELSE
			in := sd;
		END_IF;
		IF NOT in AND tx - start <= TIME_TO_UDINT2(T1) THEN
			Y := Y_start + step2;
			state := 0;
		ELSIF in AND tx - start >= TIME_TO_UDINT2(T2) THEN
			Y := Y_start2 + UDINT_TO_REAL(tx - start2) * s2 / speed;
		ELSIF in AND tx - start >= TIME_TO_UDINT2(T1) THEN
			Y := Y_start + UDINT_TO_REAL(tx - start - TIME_TO_UDINT2(T1)) * S1 / speed;
			start2 := tx;
			Y_start2 := Y;
		ELSIF NOT in THEN
			state := 0;
		END_IF;
	ELSIF su THEN
		state := 1;
		start := tx;
		step2 := ss;
		speed := 1000.0;
		Y_start := Y;
	ELSIF sd THEN

		state := 2;
		start := tx;
		step2 := -ss;
		speed := -1000.0;
		Y_start := Y;
	END_IF;

END_FUNCTION_BLOCK

PROGRAM program0
  	VAR
		SET :	BOOL;
		SU :	BOOL;
		SD :	BOOL;
		RST :	BOOL;
		SS :	REAL := 0.1;
		LIMIT_L :	REAL;
		LIMIT_H :	REAL := 100.0;
		RST_VAL :	REAL;
		SET_VAL :	REAL := 100.0;
		T1 :	TIME := T#500ms;
		T2 :	TIME := T#2s;
		S1 :	REAL := 2.0;
		S2 :	REAL := 10.0;
		Y :	REAL;
		func_block : TUNE_Block;
  	END_VAR
	func_block.SET := SET;
	func_block.SU := SU;
	func_block.SD := SD;
	func_block.RST := RST;
	func_block.SS:= SS;
	func_block.LIMIT_L := LIMIT_L;
	func_block.LIMIT_H := LIMIT_H;
	func_block.RST_VAL := RST_VAL;
	func_block.SET_VAL := SET_VAL;
	func_block.T1 := T1;
	func_block.T2 := T2;
	func_block.S1 := S1;
	func_block.S2 := S2;
	func_block();
	Y := func_block.Y;
END_PROGRAM

CONFIGURATION Config0
	VAR_GLOBAL
		PLC_TICKS_PER_SEC :	INT;
		PLC_SYS_TICK_CNT :	DINT;
	END_VAR
	RESOURCE Res0 ON PLC
		TASK task0(INTERVAL := T#20ms,PRIORITY := 0);
		PROGRAM instance0 WITH task0 : program0;
	END_RESOURCE
END_CONFIGURATION

(* ---- TUNE2.ST ---- *)
FUNCTION_BLOCK T_PLC_MS_block
	VAR_OUTPUT
		T_PLC_MS :	UDINT;
	END_VAR

	VAR_EXTERNAL
		PLC_TICKS_PER_SEC :	INT;
		PLC_SYS_TICK_CNT :	DINT;
	END_VAR

	VAR
		debug :	BOOL;(*Debug-Mode ON / OFF*)
		N :	INT;(*Debug-Faktor*)
		Offset :	UDINT;(*Debug-Offset*)
		temp :	DWORD := DWORD#1;(*Debug-Offset*)
		mode :	BOOL;(*modus*)
		faktor :	UDINT;(*Systemtakt-Faktor*)
		init :	BOOL;
		v_plc_ticks_per_sec :	UDINT;
		base :	UDINT := UDINT#1000;
	END_VAR

	IF init = FALSE THEN
		v_plc_ticks_per_sec := INT_TO_UDINT(PLC_TICKS_PER_SEC);
		IF v_plc_ticks_per_sec = UDINT#1024 THEN
			faktor := UDINT#1;
			mode := FALSE;
		ELSIF v_plc_ticks_per_sec > UDINT#0 THEN
			IF v_plc_ticks_per_sec <= base THEN
				faktor := base / v_plc_ticks_per_sec;
				mode := FALSE;
			ELSE
				faktor := v_plc_ticks_per_sec / base;
				mode := TRUE;
			END_IF;
		ELSE
			faktor := UDINT#1;
		END_IF;
		init := TRUE;
	END_IF;

	IF mode THEN
		T_PLC_MS := DINT_TO_UDINT(PLC_SYS_TICK_CNT) / faktor;
	ELSE
		T_PLC_MS := DINT_TO_UDINT(PLC_SYS_TICK_CNT) * faktor;
	END_IF;

	IF debug THEN
		T_PLC_MS := (DWORD_TO_UDINT(SHL(UDINT_TO_DWORD(T_PLC_MS),N) OR SHL(temp,N)) - UDINT#1) + Offset;
	END_IF;
END_FUNCTION_BLOCK

FUNCTION TIME_TO_UDINT2:UDINT
	VAR_INPUT
		X :	TIME;
	END_VAR

	TIME_TO_UDINT2 := DINT_TO_UDINT(TIME_TO_DINT(X));
END_FUNCTION

FUNCTION_BLOCK TUNE2_Block

	VAR_INPUT
		SET :	BOOL;
		SU :	BOOL;
		SD :	BOOL;
		FU :	BOOL;
		FD :	BOOL;
		RST :	BOOL;
		SS :	REAL := 0.1;
		FS :	REAL := 5.0;
		LIMIT_L :	REAL;
		LIMIT_H :	REAL := 100.0;
		RST_VAL :	REAL;
		SET_VAL :	REAL := 100.0;
		TR :	TIME := T#500ms;
		S1 :	REAL := 2.0;
		S2 :	REAL := 10.0;
	END_VAR

	VAR_OUTPUT
		Y :	REAL;
	END_VAR

	VAR
		tx :	UDINT;
		start :	UDINT;
		state :	INT;
		in :	BOOL;
		step2 :	REAL;
		speed :	REAL;
		Y_start :	REAL;
		T_PLC_MS :	T_PLC_MS_block;
	END_VAR

	T_PLC_MS();
	tx:= T_PLC_MS.T_PLC_MS;

	IF rst THEN
		Y := RST_val;
		state := 0;
	ELSIF set THEN
		Y := SET_val;
		state := 0;
	ELSIF state > 0 THEN
		CASE state OF
			1 :
				in := su;
			2 :
				in := sd;
			3 :
				in := fu;
			4 :
				in := fd;
		END_CASE;
		IF NOT in AND tx - start <= TIME_TO_UDINT2(TR) THEN
			Y := Y_start + step2;
			state := 0;
		ELSIF in AND tx - start >= TIME_TO_UDINT2(TR) THEN
			Y := Y_start + UDINT_TO_REAL(tx - start - TIME_TO_UDINT2(TR)) * speed;
		ELSIF NOT in THEN
			state := 0;
		END_IF;
	ELSIF su THEN
		state := 1;
		start := tx;
		step2 := ss;
		speed := s1 * 1.0E-3;
		Y_start := Y;
	ELSIF sd THEN
		state := 2;
		start := tx;
		step2 := -ss;
		speed := -s1 * 1.0E-3;
		Y_start := Y;
	ELSIF fu THEN
		state := 3;
		start := tx;
		step2 := fs;
		speed := s2 * 1.0E-3;
		y_start := Y;
	ELSIF fd THEN
		state := 4;
		start := tx;
		step2 := -fs;
		speed := -s2 * 1.0E-3;
		y_start := Y;
	END_IF;
END_FUNCTION_BLOCK

PROGRAM program0
  	VAR
		SET :	BOOL;
		SU :	BOOL;
		SD :	BOOL;
		FU :	BOOL;
		FD :	BOOL;
		RST :	BOOL;
		SS :	REAL;
		FS :	REAL;
		LIMIT_L :	REAL;
		LIMIT_H :	REAL;
		RST_VAL :	REAL;
		SET_VAL :	REAL;
		TR :	TIME ;
		S1 :	REAL;
		S2 :	REAL;
		Y :	REAL;
		func_block : TUNE2_Block;
  	END_VAR
	func_block.SET := SET;
	func_block.SU := SU;
	func_block.SD := SD;
	func_block.FU := FU;
	func_block.FD := FD;
	func_block.RST := RST;
	func_block.SS:= SS;
	func_block.FS := FS;
	func_block.LIMIT_L := LIMIT_L;
	func_block.LIMIT_H := LIMIT_H;
	func_block.RST_VAL := RST_VAL;
	func_block.SET_VAL := SET_VAL;
	func_block.TR := TR;
	func_block.S1 := S1;
	func_block.S2 := S2;
	func_block();
	Y := func_block.Y;
END_PROGRAM

CONFIGURATION Config0
	VAR_GLOBAL
		PLC_TICKS_PER_SEC :	INT;
		PLC_SYS_TICK_CNT :	DINT;
	END_VAR

	RESOURCE Res0 ON PLC
		TASK task0(INTERVAL := T#20ms,PRIORITY := 0);
		PROGRAM instance0 WITH task0 : program0;
	END_RESOURCE
END_CONFIGURATION

(* ---- URL_TO_STRING.ST ---- *)
TYPE
  oscat_STRING3               : STRING;
  oscat_STRING8               : STRING;
  oscat_STRING10              : STRING;
  oscat_STRING40              : STRING;
  oscat_STRING32              : STRING;
  oscat_STRING80              : STRING;
  oscat_STRING160              : STRING;
  oscat_STRING250              : STRING;
END_TYPE

TYPE oscat_url :
	STRUCT
		PROTOCOL : oscat_STRING10;
		USER     : oscat_STRING32;
		PASSWORD : oscat_STRING32;
		DOMAIN   : oscat_STRING80;
		PORT     : WORD;
		PATH     : oscat_STRING80;
		QUERY    : oscat_STRING250;
		ANCHOR   : oscat_STRING40;
		HEADER   : oscat_STRING160;
	END_STRUCT;
END_TYPE

FUNCTION_BLOCK URL_TO_STRING_Block

	VAR_INPUT
		IN :	oscat_url;
	END_VAR

	VAR_OUTPUT
		URL_TO_STRING :	oscat_STRING250;
	END_VAR

	IF NE_STRING(IN.PROTOCOL,'') THEN URL_TO_STRING := CONCAT(IN.PROTOCOL,'://'); END_IF;

	IF NE_STRING(IN.USER,'') THEN
		URL_TO_STRING := CONCAT(URL_TO_STRING, IN.USER);
		IF NE_STRING(IN.PASSWORD,'') THEN
			URL_TO_STRING := CONCAT(URL_TO_STRING, ':');
			URL_TO_STRING := CONCAT(URL_TO_STRING, IN.PASSWORD);
		END_IF;
		URL_TO_STRING := CONCAT(URL_TO_STRING, '@');
	END_IF;

	URL_TO_STRING := CONCAT(URL_TO_STRING, IN.DOMAIN);

	IF IN.PORT > WORD#0 THEN
		URL_TO_STRING := CONCAT(URL_TO_STRING, ':');
		URL_TO_STRING := CONCAT(URL_TO_STRING, WORD_TO_STRING(IN.PORT));
	END_IF;

	URL_TO_STRING := CONCAT(URL_TO_STRING, IN.PATH);

	IF NE_STRING(IN.QUERY,'') THEN
		URL_TO_STRING := CONCAT(URL_TO_STRING, '?');
		URL_TO_STRING := CONCAT(URL_TO_STRING, IN.QUERY);
	END_IF;

	IF NE_STRING(IN.ANCHOR,'') THEN
		URL_TO_STRING := CONCAT(URL_TO_STRING, '#');
		URL_TO_STRING := CONCAT(URL_TO_STRING, IN.ANCHOR);
	END_IF;

END_FUNCTION_BLOCK

PROGRAM program0
	VAR
		IN :	oscat_url;
		URL_TO_STRING :	oscat_STRING250;

		func_block : URL_TO_STRING_Block;
	END_VAR
	func_block.IN := IN;

	func_block();
	URL_TO_STRING  := func_block.URL_TO_STRING;
END_PROGRAM

CONFIGURATION Config0
	RESOURCE Res0 ON PLC
		TASK task0(INTERVAL := T#20ms,PRIORITY := 0);
		PROGRAM instance0 WITH task0 : program0;
	END_RESOURCE
END_CONFIGURATION

(* ---- V3_ABS.ST ---- *)
TYPE oscat_vector_3:
	STRUCT
		X : REAL;
		Y : REAL;
		Z : REAL;
	END_STRUCT;
END_TYPE

FUNCTION_BLOCK V3_ABS_Block

	VAR_INPUT
		A :	oscat_vector_3;
	END_VAR

	VAR_OUTPUT
		V3_ABS :	REAL;
	END_VAR

	V3_ABS := SQRT(A.X * A.X + A.Y * A.Y + A.Z * A.Z);

END_FUNCTION_BLOCK

PROGRAM program0
  	VAR
		A :	oscat_vector_3;
		V3_ABS :	REAL;
		func_block : V3_ABS_Block;
  	END_VAR
	func_block.A := A;
	func_block();
	V3_ABS := func_block.V3_ABS;
END_PROGRAM

CONFIGURATION Config0
	RESOURCE Res0 ON PLC
		TASK task0(INTERVAL := T#20ms,PRIORITY := 0);
		PROGRAM instance0 WITH task0 : program0;
	END_RESOURCE
END_CONFIGURATION

(* ---- V3_ADD.ST ---- *)
TYPE oscat_vector_3:
	STRUCT
		X : REAL;
		Y : REAL;
		Z : REAL;
	END_STRUCT;
END_TYPE

FUNCTION_BLOCK V3_ADD_Block
	VAR_INPUT
		A :	oscat_vector_3;
		B :	oscat_vector_3;
	END_VAR

	VAR_OUTPUT
		V3_ADD :	oscat_vector_3;
	END_VAR

	V3_ADD.X := A.X + B.X;
	V3_ADD.Y := A.Y + B.Y;
	V3_ADD.Z := A.Z + B.Z;

END_FUNCTION_BLOCK

PROGRAM program0
  	VAR
		A :	oscat_vector_3;
		B :	oscat_vector_3;
		V3_ADD :	oscat_vector_3;
		func_block : V3_ADD_Block;
  	END_VAR
	func_block.A := A;
	func_block.B := B;
	func_block();
	V3_ADD := func_block.V3_ADD;
END_PROGRAM

CONFIGURATION Config0
  RESOURCE Res0 ON PLC
    TASK task0(INTERVAL := T#20ms,PRIORITY := 0);
    PROGRAM instance0 WITH task0 : program0;
  END_RESOURCE
END_CONFIGURATION

(* ---- V3_ANG.ST ---- *)
TYPE oscat_vector_3:
	STRUCT
		X : REAL;
		Y : REAL;
		Z : REAL;
	END_STRUCT;
END_TYPE

FUNCTION_BLOCK V3_ABS_Block
	VAR_INPUT
		A :	oscat_vector_3;
	END_VAR

	VAR_OUTPUT
		V3_ABS : REAL;
	END_VAR

	V3_ABS := SQRT(A.X * A.X + A.Y * A.Y + A.Z * A.Z);

END_FUNCTION_BLOCK

FUNCTION_BLOCK V3_DPRO_Block

	VAR_INPUT
		A :	oscat_vector_3;
		B :	oscat_vector_3;
	END_VAR

	VAR_OUTPUT
		V3_DPRO :	REAL;
	END_VAR

	V3_DPRO := A.X * B.X + A.Y * B.Y + A.Z * B.Z;

END_FUNCTION_BLOCK

FUNCTION_BLOCK V3_ANG_Block

	VAR_INPUT
		A :	oscat_vector_3;
		B :	oscat_vector_3;
	END_VAR

	VAR_OUTPUT
		V3_ANG :	REAL;
	END_VAR

	VAR
		d :	REAL;
		V3_ABS :	V3_ABS_Block;
		V3_DPRO :	V3_DPRO_Block;
	END_VAR

	V3_ABS(A:=A);
	d :=V3_ABS.V3_ABS;

	V3_ABS(A:=B);
	d := d * V3_ABS.V3_ABS;

	IF d > 0.0 THEN
		V3_DPRO(A:=A,B:=B);
		V3_ANG := ACOS(LIMIT(-1.0, V3_DPRO.V3_DPRO / d,1.0));
	ELSE
		V3_ANG := 0.0;

	END_IF;

END_FUNCTION_BLOCK

PROGRAM program0
  	VAR
		A :	oscat_vector_3;
		B :	oscat_vector_3;
		V3_ANG :	REAL;
		func_block : V3_ANG_Block;
  	END_VAR
	func_block.A := A;
	func_block.B := B;
	func_block();
	V3_ANG := func_block.V3_ANG;
END_PROGRAM

CONFIGURATION Config0
  RESOURCE Res0 ON PLC
    TASK task0(INTERVAL := T#20ms,PRIORITY := 0);
    PROGRAM instance0 WITH task0 : program0;
  END_RESOURCE
END_CONFIGURATION

(* ---- V3_DPRO.ST ---- *)
TYPE oscat_vector_3:
	STRUCT
		X : REAL;
		Y : REAL;
		Z : REAL;
	END_STRUCT;
END_TYPE

FUNCTION_BLOCK V3_DPRO_Block

	VAR_INPUT
		A :	oscat_vector_3;
		B :	oscat_vector_3;
	END_VAR

	VAR_OUTPUT
		V3_DPRO :	REAL;
	END_VAR

	V3_DPRO := A.X * B.X + A.Y * B.Y + A.Z * B.Z;

END_FUNCTION_BLOCK

PROGRAM program0
  	VAR
		A :	oscat_vector_3;
		B :	oscat_vector_3;
		V3_DPRO : REAL;
		func_block : V3_DPRO_Block;
  	END_VAR
	func_block.A := A;
	func_block.B := B;
	func_block();
	V3_DPRO := func_block.V3_DPRO;
END_PROGRAM

CONFIGURATION Config0
  RESOURCE Res0 ON PLC
    TASK task0(INTERVAL := T#20ms,PRIORITY := 0);
    PROGRAM instance0 WITH task0 : program0;
  END_RESOURCE
END_CONFIGURATION

(* ---- V3_NORM.ST ---- *)
TYPE oscat_vector_3:
	STRUCT
		X : REAL;
		Y : REAL;
		Z : REAL;
	END_STRUCT;
END_TYPE

FUNCTION_BLOCK V3_ABS_Block

	VAR_INPUT
		A :	oscat_vector_3;
	END_VAR

	VAR_OUTPUT
		V3_ABS :	REAL;
	END_VAR

	V3_ABS := SQRT(A.X * A.X + A.Y * A.Y + A.Z * A.Z);

END_FUNCTION_BLOCK

FUNCTION_BLOCK V3_SMUL_Block
	VAR_INPUT
		A :	oscat_vector_3;
		M :	REAL;
	END_VAR

	VAR_OUTPUT
		V3_SMUL :	oscat_vector_3;
	END_VAR

	V3_SMUL.X := A.X * M;
	V3_SMUL.Y := A.Y * M;
	V3_SMUL.Z := A.Z * M;
END_FUNCTION_BLOCK

FUNCTION_BLOCK V3_NORM_Block

	VAR_INPUT
		A :	oscat_vector_3;
	END_VAR

	VAR_OUTPUT
		V3_NORM :	oscat_vector_3;
	END_VAR

	VAR
		la :	REAL;
		V3_SMUL :	V3_SMUL_Block;
		V3_ABS :	V3_ABS_Block;
	END_VAR

	V3_ABS(A:=A);
	la:=V3_ABS.V3_ABS;

	IF la > 0.0 THEN
		V3_SMUL(A:=A,M:=1.0/la);
		V3_NORM:=V3_SMUL.V3_SMUL;
	ELSE
		V3_NORM.X := 0.0;
		V3_NORM.Y := 0.0;
		V3_NORM.Z := 0.0;
	END_IF;

END_FUNCTION_BLOCK

PROGRAM program0
  	VAR
		A :	oscat_vector_3;
		V3_NORM :	oscat_vector_3;
		func_block : V3_NORM_Block;
  	END_VAR
	func_block.A := A;
	func_block();
	V3_NORM := func_block.V3_NORM;
END_PROGRAM

CONFIGURATION Config0
  RESOURCE Res0 ON PLC
    TASK task0(INTERVAL := T#20ms,PRIORITY := 0);
    PROGRAM instance0 WITH task0 : program0;
  END_RESOURCE
END_CONFIGURATION

(* ---- V3_NUL.ST ---- *)
TYPE oscat_vector_3:
	STRUCT
		X : REAL;
		Y : REAL;
		Z : REAL;
	END_STRUCT;
END_TYPE

FUNCTION_BLOCK V3_NUL_Block

	VAR_INPUT
		A :	oscat_vector_3;
	END_VAR

	VAR_OUTPUT
		V3_NUL :	BOOL;
	END_VAR

	V3_NUL := A.X = 0.0 AND A.Y = 0.0 AND A.Z = 0.0;

END_FUNCTION_BLOCK

PROGRAM program0
  	VAR
		A :	oscat_vector_3;
		V3_NUL :	BOOL;
		func_block : V3_NUL_Block;
  	END_VAR
	func_block.A := A;
	func_block();
	V3_NUL := func_block.V3_NUL;
END_PROGRAM

CONFIGURATION Config0
  RESOURCE Res0 ON PLC
    TASK task0(INTERVAL := T#20ms,PRIORITY := 0);
    PROGRAM instance0 WITH task0 : program0;
  END_RESOURCE
END_CONFIGURATION

(* ---- V3_PAR.ST ---- *)
TYPE oscat_vector_3:
	STRUCT
		X : REAL;
		Y : REAL;
		Z : REAL;
	END_STRUCT;
END_TYPE

FUNCTION_BLOCK V3_ABS_Block

	VAR_INPUT
		A :	oscat_vector_3;
	END_VAR

	VAR_OUTPUT
		V3_ABS :	REAL;
	END_VAR

	V3_ABS := SQRT(A.X * A.X + A.Y * A.Y + A.Z * A.Z);

END_FUNCTION_BLOCK

FUNCTION_BLOCK V3_XPRO_Block
	VAR_INPUT
		A :	oscat_vector_3;
		B :	oscat_vector_3;
	END_VAR

	VAR_OUTPUT
		V3_XPRO :	oscat_vector_3;
	END_VAR

	V3_XPRO.X := A.Y * B.Z - A.Z * B.Y;
	V3_XPRO.Y := A.Z * B.X - A.X * B.Z;
	V3_XPRO.Z := A.X * B.Y - A.Y * B.X;

END_FUNCTION_BLOCK

FUNCTION_BLOCK V3_PAR_Block
	VAR_INPUT
		A :	oscat_vector_3;
		B :	oscat_vector_3;
	END_VAR

	VAR_OUTPUT
		V3_PAR :	BOOL;
	END_VAR

	VAR
		V3_XPRO :	V3_XPRO_Block;
		V3_ABS :	V3_ABS_Block;
	END_VAR

	V3_XPRO(A:=A,B:=B);
	V3_ABS(A:=V3_XPRO.V3_XPRO);

	V3_PAR := V3_ABS.V3_ABS = 0.0;

END_FUNCTION_BLOCK

PROGRAM program0
  	VAR
		A :	oscat_vector_3;
		B :	oscat_vector_3;
		V3_PAR :	BOOL;
		func_block : V3_PAR_Block;
  	END_VAR
	func_block.A := A;
	func_block.B := B;
	func_block();
	V3_PAR := func_block.V3_PAR;
END_PROGRAM

CONFIGURATION Config0
  RESOURCE Res0 ON PLC
    TASK task0(INTERVAL := T#20ms,PRIORITY := 0);
    PROGRAM instance0 WITH task0 : program0;
  END_RESOURCE
END_CONFIGURATION

(* ---- V3_REV.ST ---- *)
TYPE oscat_vector_3:
	STRUCT
		X : REAL;
		Y : REAL;
		Z : REAL;
	END_STRUCT;
END_TYPE

FUNCTION_BLOCK V3_REV_Block
	VAR_INPUT
		A :	oscat_vector_3;
	END_VAR

	VAR_OUTPUT
		V3_REV :	oscat_vector_3;
	END_VAR

	V3_REV.X := -A.X;
	V3_REV.Y := -A.Y;
	V3_REV.Z := -A.Z;

END_FUNCTION_BLOCK

PROGRAM program0
  	VAR
		A :	oscat_vector_3;
		V3_REV : oscat_vector_3;
		func_block : V3_REV_Block;
  	END_VAR
	func_block.A := A;
	func_block();
	V3_REV := func_block.V3_REV;
END_PROGRAM

CONFIGURATION Config0
  RESOURCE Res0 ON PLC
    TASK task0(INTERVAL := T#20ms,PRIORITY := 0);
    PROGRAM instance0 WITH task0 : program0;
  END_RESOURCE
END_CONFIGURATION

(* ---- V3_SMUL.ST ---- *)
TYPE oscat_vector_3:
	STRUCT
		X : REAL;
		Y : REAL;
		Z : REAL;
	END_STRUCT;
END_TYPE

FUNCTION_BLOCK V3_SMUL_Block
	VAR_INPUT
		A :	oscat_vector_3;
		M :	REAL;
	END_VAR

	VAR_OUTPUT
		V3_SMUL :	oscat_vector_3;
	END_VAR

	V3_SMUL.X := A.X * M;
	V3_SMUL.Y := A.Y * M;
	V3_SMUL.Z := A.Z * M;
END_FUNCTION_BLOCK

PROGRAM program0
  	VAR
		A :	oscat_vector_3;
		M :	REAL;
		V3_SMUL :	oscat_vector_3;
		func_block : V3_SMUL_Block;
  	END_VAR
	func_block.A := A;
	func_block.M := M;
	func_block();
	V3_SMUL := func_block.V3_SMUL;
END_PROGRAM

CONFIGURATION Config0
	RESOURCE Res0 ON PLC
		TASK task0(INTERVAL := T#20ms,PRIORITY := 0);
		PROGRAM instance0 WITH task0 : program0;
	END_RESOURCE
END_CONFIGURATION

(* ---- V3_SUB.ST ---- *)
TYPE oscat_vector_3:
	STRUCT
		X : REAL;
		Y : REAL;
		Z : REAL;
	END_STRUCT;
END_TYPE

FUNCTION_BLOCK V3_SUB_Block

	VAR_INPUT
		A :	oscat_vector_3;
		B :	oscat_vector_3;
	END_VAR

	VAR_OUTPUT
		V3_SUB :	oscat_vector_3;
	END_VAR

	V3_SUB.X := A.X - B.X;
	V3_SUB.Y := A.Y - B.Y;
	V3_SUB.Z := A.Z - B.Z;

END_FUNCTION_BLOCK

PROGRAM program0
  	VAR
		A :	oscat_vector_3;
		B :	oscat_vector_3;
		V3_SUB :	oscat_vector_3;
		func_block : V3_SUB_Block;
  	END_VAR
	func_block.A := A;
	func_block.B := B;
	func_block();
	V3_SUB := func_block.V3_SUB;
END_PROGRAM

CONFIGURATION Config0
  RESOURCE Res0 ON PLC
    TASK task0(INTERVAL := T#20ms,PRIORITY := 0);
    PROGRAM instance0 WITH task0 : program0;
  END_RESOURCE
END_CONFIGURATION

(* ---- V3_XANG.ST ---- *)
TYPE oscat_vector_3 :
	STRUCT
		X : REAL;
		Y : REAL;
		Z : REAL;
	END_STRUCT;
END_TYPE

FUNCTION_BLOCK V3_ABS_Block

	VAR_INPUT
		A :	oscat_vector_3;
	END_VAR

	VAR_OUTPUT
		V3_ABS :	REAL;
	END_VAR

	V3_ABS := SQRT(A.X * A.X + A.Y * A.Y + A.Z * A.Z);

END_FUNCTION_BLOCK

FUNCTION_BLOCK V3_XANG_Block

	VAR_INPUT
		A :	oscat_vector_3;
	END_VAR

	VAR_OUTPUT
		V3_XANG :	REAL;
	END_VAR

	VAR
		la :	REAL;
		V3_ABS :	V3_ABS_Block;
	END_VAR

	V3_ABS(A:=A);
	la:=V3_ABS.V3_ABS;

	IF la > 0.0 THEN
		V3_XANG := ACOS(A.X / la);
	ELSE
		V3_XANG := 0.0;
	END_IF;

END_FUNCTION_BLOCK

PROGRAM program0
  	VAR
		A :	oscat_vector_3;
		V3_XANG :	REAL;
		func_block : V3_XANG_Block;
  	END_VAR
	func_block.A := A;
	func_block();
	V3_XANG := func_block.V3_XANG;
END_PROGRAM

CONFIGURATION Config0
  RESOURCE Res0 ON PLC
    TASK task0(INTERVAL := T#20ms,PRIORITY := 0);
    PROGRAM instance0 WITH task0 : program0;
  END_RESOURCE
END_CONFIGURATION

(* ---- V3_XPRO.ST ---- *)
TYPE oscat_vector_3 :
	STRUCT
		X : REAL;
		Y : REAL;
		Z : REAL;
	END_STRUCT;
END_TYPE

FUNCTION_BLOCK V3_XPRO_Block
	VAR_INPUT
		A :	oscat_vector_3;
		B :	oscat_vector_3;
	END_VAR

	VAR_OUTPUT
		V3_XPRO :	oscat_vector_3;
	END_VAR

	V3_XPRO.X := A.Y * B.Z - A.Z * B.Y;
	V3_XPRO.Y := A.Z * B.X - A.X * B.Z;
	V3_XPRO.Z := A.X * B.Y - A.Y * B.X;

END_FUNCTION_BLOCK

PROGRAM program0
  	VAR
		A :	oscat_vector_3;
		B :	oscat_vector_3;
		V3_XPRO :	oscat_vector_3;
		func_block : V3_XPRO_Block;
  	END_VAR
	func_block.A := A;
	func_block.B := B;
	func_block();
	V3_XPRO := func_block.V3_XPRO;
END_PROGRAM

CONFIGURATION Config0
  RESOURCE Res0 ON PLC
    TASK task0(INTERVAL := T#20ms,PRIORITY := 0);
    PROGRAM instance0 WITH task0 : program0;
  END_RESOURCE
END_CONFIGURATION

(* ---- V3_YANG.ST ---- *)
TYPE oscat_vector_3:
  	STRUCT
		X : REAL;
		Y : REAL;
		Z : REAL;
  	END_STRUCT;
END_TYPE

FUNCTION_BLOCK V3_ABS_Block

	VAR_INPUT
		A :	oscat_vector_3;
	END_VAR

	VAR_OUTPUT
		V3_ABS :	REAL;
	END_VAR

	V3_ABS := SQRT(A.X * A.X + A.Y * A.Y + A.Z * A.Z);

END_FUNCTION_BLOCK

FUNCTION_BLOCK V3_YANG_Block
	VAR_INPUT
		A :	oscat_vector_3;
	END_VAR

	VAR_OUTPUT
		V3_YANG :	REAL;
	END_VAR

	VAR
		la :	REAL;
		V3_ABS :	V3_ABS_Block;
	END_VAR

	V3_ABS(A:=A);
	la:=V3_ABS.V3_ABS;

	IF la > 0.0 THEN
		V3_YANG := ACOS(A.Y / la);
	ELSE
		V3_YANG := 0.0;
	END_IF;

END_FUNCTION_BLOCK

PROGRAM program0
  	VAR
		A :	oscat_vector_3;
		V3_YANG :	REAL;
		func_block : V3_YANG_Block;
  	END_VAR
	func_block.A := A;
	func_block();
	V3_YANG := func_block.V3_YANG;
END_PROGRAM

CONFIGURATION Config0
  RESOURCE Res0 ON PLC
    TASK task0(INTERVAL := T#20ms,PRIORITY := 0);
    PROGRAM instance0 WITH task0 : program0;
  END_RESOURCE
END_CONFIGURATION

(* ---- V3_ZANG.ST ---- *)
TYPE oscat_vector_3:
  STRUCT
	X : REAL;
	Y : REAL;
	Z : REAL;
  END_STRUCT;
END_TYPE

FUNCTION_BLOCK V3_ABS_Block

	VAR_INPUT
		A :	oscat_vector_3;
	END_VAR

	VAR_OUTPUT
		V3_ABS :	REAL;
	END_VAR

	V3_ABS := SQRT(A.X * A.X + A.Y * A.Y + A.Z * A.Z);

END_FUNCTION_BLOCK

FUNCTION_BLOCK V3_ZANG_Block
	VAR_INPUT
		A :	oscat_vector_3;
	END_VAR

	VAR_OUTPUT
		V3_ZANG :	REAL;
	END_VAR

	VAR
		la :	REAL;
		V3_ABS :	V3_ABS_Block;
	END_VAR

	V3_ABS(A:=A);
	la:=V3_ABS.V3_ABS;

	IF la > 0.0 THEN
		V3_ZANG := ACOS(A.Z / la);
	ELSE
		V3_ZANG := 0.0;
	END_IF;

END_FUNCTION_BLOCK

PROGRAM program0
  	VAR
		A :	oscat_vector_3;
		V3_ZANG :	REAL;
		func_block : V3_ZANG_Block;
  	END_VAR
	func_block.A := A;
	func_block();
	V3_ZANG := func_block.V3_ZANG;
END_PROGRAM

CONFIGURATION Config0
  RESOURCE Res0 ON PLC
    TASK task0(INTERVAL := T#20ms,PRIORITY := 0);
    PROGRAM instance0 WITH task0 : program0;
  END_RESOURCE
END_CONFIGURATION

(* ---- WATER_CP.ST ---- *)
TYPE
	oscat_ARRAY_X               : ARRAY [0..1]    OF REAL;
	oscat_XY                    : ARRAY [1..20]   OF oscat_ARRAY_X := [0,0,0,0,0,0,0,0,0,0,0,0,0,0,0,0,0,0,0,0];
END_TYPE

FUNCTION_BLOCK LINEAR_INT_Block

	VAR_INPUT
		X :	REAL;
		XY :	oscat_XY;
		PTS :	INT;
	END_VAR

	VAR_OUTPUT
		LINEAR_INT :	REAL;
	END_VAR

	VAR
		i :	INT;
		i2 :	INT;
	END_VAR

	pts := MIN(pts,20);

	i := 2;

	WHILE (i < pts) AND (XY[i][0] < X) DO
		i := i + 1;
	END_WHILE;

	i2 := i-1;

	LINEAR_INT := ((XY[i][1] - XY[i2][1]) * X - XY[i][1] * XY[i2][0] + XY[i2][1] * XY[i][0]) / (XY[i][0] - XY[i2][0]);

END_FUNCTION_BLOCK

FUNCTION_BLOCK WATER_CP_Block

    VAR_INPUT
        T :	REAL;
    END_VAR

    VAR_OUTPUT
        CAP :	REAL;
    END_VAR

    VAR
        Pts :	INT;
        data :	oscat_XY;
        FB_LINEAR_INT :	LINEAR_INT_Block;
    END_VAR

    IF Pts = 0 THEN
        Pts := 10;

        data[01][0] := REAL#0.0;
        data[01][1] := REAL#4.228;
        data[02][0] := REAL#05.0;
        data[02][1] := REAL#4.200;
        data[03][0] := REAL#10.0;
        data[03][1] := REAL#4.188;
        data[04][0] := REAL#15.0;
        data[04][1] := REAL#4.184;
        data[05][0] := REAL#50.0;
        data[05][1] := REAL#4.181;
        data[06][0] := REAL#60.0;
        data[06][1] := REAL#4.183;
        data[07][0] := REAL#70.0;
        data[07][1] := REAL#4.187;
        data[08][0] := REAL#80.0;
        data[08][1] := REAL#4.194;
        data[09][0] := REAL#90.0;
        data[09][1] := REAL#4.204;
        data[10][0] := REAL#100.0;
        data[10][1] := REAL#4.220;

    END_IF;

    FB_LINEAR_INT(X:=T,XY:=Data,Pts:=Pts);
    cap:=FB_LINEAR_INT.LINEAR_INT;

END_FUNCTION_BLOCK

PROGRAM program0
	VAR
		T :	REAL;
        CAP :	REAL;

		func_block : WATER_CP_Block;
	END_VAR
	func_block.T := T;

	func_block();
	CAP  := func_block.CAP;
END_PROGRAM

CONFIGURATION Config0
	RESOURCE Res0 ON PLC
		TASK task0(INTERVAL := T#20ms,PRIORITY := 0);
		PROGRAM instance0 WITH task0 : program0;
	END_RESOURCE
END_CONFIGURATION

(* ---- WATER_ENTHALPY.ST ---- *)
TYPE
	oscat_ARRAY_X               : ARRAY [0..1]    OF REAL;
	oscat_XY                    : ARRAY [1..20]   OF oscat_ARRAY_X := [0,0,0,0,0,0,0,0,0,0,0,0,0,0,0,0,0,0,0,0];
END_TYPE

FUNCTION_BLOCK LINEAR_INT_Block

	VAR_INPUT
		X :	REAL;
		XY :	oscat_XY;
		PTS :	INT;
	END_VAR

	VAR_OUTPUT
		LINEAR_INT :	REAL;
	END_VAR

	VAR
		i :	INT;
		i2 :	INT;
	END_VAR

	pts := MIN(pts,20);

	i := 2;

	WHILE (i < pts) AND (XY[i][0] < X) DO
		i := i + 1;
	END_WHILE;

	i2 := i-1;

	LINEAR_INT := ((XY[i][1] - XY[i2][1]) * X - XY[i][1] * XY[i2][0] + XY[i2][1] * XY[i][0]) / (XY[i][0] - XY[i2][0]);

END_FUNCTION_BLOCK

FUNCTION_BLOCK WATER_ENTHALPY_Block

    VAR_INPUT
        T :	REAL;
    END_VAR

    VAR_OUTPUT
        RESULT :	REAL;
    END_VAR

    VAR
        Pts :	INT;
        data :	oscat_XY;
        FB_LINEAR_INT :	LINEAR_INT_Block;
    END_VAR

    IF Pts = 0 THEN
        Pts := 11;
        data[01][0] := REAL#0.0;
        data[01][1] := REAL#0.06;
        data[02][0] := REAL#10.0;
        data[02][1] := REAL#42.1;
        data[03][0] := REAL#20.0;
        data[03][1] := REAL#83.9;
        data[04][0] := REAL#30.0;
        data[04][1] := REAL#125.8;
        data[05][0] := REAL#40.0;
        data[05][1] := REAL#167.58;
        data[06][0] := REAL#50.0;
        data[06][1] := REAL#209.4;
        data[07][0] := REAL#60.0;
        data[07][1] := REAL#251.2;
        data[08][0] := REAL#70.0;
        data[08][1] := REAL#293.1;
        data[09][0] := REAL#80.0;
        data[09][1] := REAL#335.0;
        data[10][0] := REAL#90.0;
        data[10][1] := REAL#377.0;
        data[11][0] := REAL#100.0;
        data[11][1] := REAL#419.1;
    END_IF;

    FB_LINEAR_INT(X:=T,XY:=Data,Pts:=Pts);
    Result :=FB_LINEAR_INT.LINEAR_INT;

END_FUNCTION_BLOCK

PROGRAM program0
	VAR
		T :	REAL;
		RESULT :	REAL;

		func_block : WATER_ENTHALPY_Block;
	END_VAR
	func_block.T := T;

	func_block();
	RESULT  := func_block.RESULT;
END_PROGRAM

CONFIGURATION Config0
	RESOURCE Res0 ON PLC
		TASK task0(INTERVAL := T#20ms,PRIORITY := 0);
		PROGRAM instance0 WITH task0 : program0;
	END_RESOURCE
END_CONFIGURATION

(* ---- WORLD_WEATHER_DESC_GE.ST ---- *)
TYPE
  oscat_STRING3               : STRING;
  oscat_STRING8               : STRING;
  oscat_STRING10              : STRING;
  oscat_STRING60              : STRING;
END_TYPE

TYPE
	oscat_WORLD_WEATHER_CUR :
	STRUCT
		OBSERVATION_TIME : oscat_STRING8;
		TEMP_C           : INT;
		WEATHER_CODE     : INT;
		WEATHER_DESC 	 : oscat_STRING60;
		WEATHER_ICON     : INT;
		WIND_SPEED_MILES : INT;
		WIND_SPEED_KMPH  : INT;
		WIND_DIR_DEGREE  : INT;
		WIND_DIR16POINT  : oscat_STRING3;
		PRECIPMM         : REAL;
		HUMIDITY         : INT;
		VISIBILITY       : INT;
		PRESSURE         : INT;
		CLOUDOVER        : INT;
	END_STRUCT;

	oscat_WORLD_WEATHER_DAY :
	STRUCT
		DATE_OF_DAY      : oscat_STRING10;
		TEMP_MAX_C       : INT;
		TEMP_MAX_F       : INT;
		TEMP_MIN_C       : INT;
		TEMP_MIN_F       : INT;
		WIND_SPEED_MILES : INT;
		WIND_SPEED_KMPH  : INT;
		WIND_DIR_DEGREE  : INT;
		WIND_DIR16POINT  : oscat_STRING3;
		WEATHER_CODE     : INT;
		WEATHER_DESC     : oscat_STRING60;
		WEATHER_ICON     : INT;
		PRECIPMM         : REAL;
	END_STRUCT;

	oscat_WORLD_WEATHER_DAY_ARR : ARRAY [0..4] OF oscat_WORLD_WEATHER_DAY;

	oscat_WORLD_WEATHER_DATA :
	STRUCT
		CUR : oscat_WORLD_WEATHER_CUR;
		DAY : oscat_WORLD_WEATHER_DAY_ARR;
	END_STRUCT;

	oscat_WORLD_WEATHER_aI0_41 : ARRAY[0..41] OF INT;
END_TYPE

FUNCTION_BLOCK WORLD_WEATHER_DESC_GE_Block

	VAR_INPUT
		ACTIVATE :	BOOL;
	END_VAR

	VAR_IN_OUT
		WW :	oscat_WORLD_WEATHER_DATA;
	END_VAR

	VAR
		act_last :	BOOL;
		x :	INT;
		y :	INT;
		str :	oscat_STRING60;
		i :	INT;
	END_VAR

	IF ACTIVATE AND act_last = FALSE THEN
		i := 0;
		FOR y := 1 TO 12 DO
			CASE y OF
			1,3,5,7,9:	x :=  WW.DAY[i].WEATHER_CODE;
			2,4,6,8,10:	WW.DAY[i].WEATHER_DESC := str;
						i := i + 1;
			11:			x :=  WW.CUR.WEATHER_CODE;
			12:			WW.CUR.WEATHER_DESC := str;
			END_CASE;

			CASE x OF
				113	:	str := 'heiter/sonnig';
				116	:	str := 'stellenweise wolkig';
				119	:	str := 'wolkig';
				122	:	str := 'awret';
				143	:	str := 'Nebel';
				176	:	str := 'stellenweise nahegelegener Regen';
				179	:	str := 'stellenweise nahegelegener Schneefall';
				182	:	str := 'stellenweise nahegelegener Eisregen';
				185	:	str := 'stellenweise gefrierender Niesel';
				200	:	str := 'nahegelegene Sturm';
				227	:	str := 'Schneetreiben';
				230	:	str := 'Schneesturm';
				248	:	str := 'Nebel';
				260	:	str := 'gefrierender Nebel';
				263	:	str := 'stellenweise leichter Nieselregen';
				266	:	str := 'leichter Niesel';
				281	:	str := 'gefrierender Nieselregen';
				284	:	str := 'stark gefrierender Nieselregen';
				293	:	str := 'stellenweise leichter Regen';
				296	:	str := 'leichter Regen';
				299	:	str := 'zeitweise etwas Regen';
				302	:	str := 'awerg Regen';
				305	:	str := 'zeitweise etwas starker Regen';
				308	:	str := 'starker Regen';
				311	:	str := 'leichter gefrierender Regen';
				314	:	str := 'awerawer oder starker Eisregen';
				317	:	str := 'leichter Eisregen';
				320	:	str := 'awewea oder starker Eisregen';
				323	:	str := 'stellenweise leichter Schneefall';
				326	:	str := 'leichter Scheefall';
				329	:	str := 'stellenweise moderater Schneefall';
				332	:	str := 'awertwy Schnee';
				335	:	str := 'stellenweise starker Scheefall';
				338	:	str := 'starker Schneefall';
				350	:	str := 'Hagel';
				353	:	str := 'leichte ewruerh';
				356	:	str := 'awerwaer oder starker Regenfall';
				359	:	str := 'sintflutartige aweheawh';
				362	:	str := 'leichter Eisregen';
				365	:	str := 'aweraweb oder starker Eisregen';
				368	:	str := 'leichte Schneeschauer';
				371	:	str := 'awerawb oder starker Schneefall';
				374	:	str := 'leichter Hagel';
				377	:	str := 'awerawer oder starker Hagel';
				386	:	str := 'stellenweise leichter Regen in Gewittergebiet';
				389	:	str := 'awer oder starker Regen in Gewittergebiet';
				392	:	str := 'stellenweise leichter Schneefall in Gewittergebiet';
				395	:	str := 'awerh oder starker Schnee in Gewittergebiet';
			ELSE
				str := 	'nicht aweh';
			END_CASE;
		END_FOR;
	END_IF;
	act_last := ACTIVATE;

END_FUNCTION_BLOCK

PROGRAM program0
	VAR
		ACTIVATE :	BOOL;
		WW :	oscat_WORLD_WEATHER_DATA;

		func_block : WORLD_WEATHER_DESC_GE_Block;
	END_VAR
	func_block.ACTIVATE := ACTIVATE;
	func_block.WW := WW;

	func_block();
	WW  := func_block.WW;
END_PROGRAM

CONFIGURATION Config0
	RESOURCE Res0 ON PLC
		TASK task0(INTERVAL := T#20ms,PRIORITY := 0);
		PROGRAM instance0 WITH task0 : program0;
	END_RESOURCE
END_CONFIGURATION

(* ---- WORLD_WEATHER_ICON_OSCAT.ST ---- *)
TYPE
  oscat_STRING3               : STRING;
  oscat_STRING8               : STRING;
  oscat_STRING10              : STRING;
  oscat_STRING60              : STRING;

END_TYPE
TYPE
	oscat_WORLD_WEATHER_CUR :
	STRUCT
		OBSERVATION_TIME : oscat_STRING8;
		TEMP_C           : INT;
		WEATHER_CODE     : INT;
		WEATHER_DESC 	 : oscat_STRING60;
		WEATHER_ICON     : INT;
		WIND_SPEED_MILES : INT;
		WIND_SPEED_KMPH  : INT;
		WIND_DIR_DEGREE  : INT;
		WIND_DIR16POINT  : oscat_STRING3;
		PRECIPMM         : REAL;
		HUMIDITY         : INT;
		VISIBILITY       : INT;
		PRESSURE         : INT;
		CLOUDOVER        : INT;
	END_STRUCT;

	oscat_WORLD_WEATHER_DAY :
	STRUCT
		DATE_OF_DAY      : oscat_STRING10;
		TEMP_MAX_C       : INT;
		TEMP_MAX_F       : INT;
		TEMP_MIN_C       : INT;
		TEMP_MIN_F       : INT;
		WIND_SPEED_MILES : INT;
		WIND_SPEED_KMPH  : INT;
		WIND_DIR_DEGREE  : INT;
		WIND_DIR16POINT  : oscat_STRING3;
		WEATHER_CODE     : INT;
		WEATHER_DESC     : oscat_STRING60;
		WEATHER_ICON     : INT;
		PRECIPMM         : REAL;
	END_STRUCT;

	oscat_WORLD_WEATHER_DAY_ARR : ARRAY [0..4] OF oscat_WORLD_WEATHER_DAY;

	oscat_WORLD_WEATHER_DATA :
	STRUCT
		CUR : oscat_WORLD_WEATHER_CUR;
		DAY : oscat_WORLD_WEATHER_DAY_ARR;
	END_STRUCT;

	oscat_WORLD_WEATHER_aI0_41 : ARRAY[0..41] OF INT;
END_TYPE

FUNCTION_BLOCK WORLD_WEATHER_ICON_OSCAT_Block

	VAR_INPUT
		ACTIVATE :	BOOL;
	END_VAR

	VAR_IN_OUT
		WW :	oscat_WORLD_WEATHER_DATA;
	END_VAR

	VAR
		act_last :	BOOL;
		x :	INT;
		i :	INT;
		init :	BOOL;
		dat :	oscat_WORLD_WEATHER_aI0_41;
	END_VAR

	IF not init THEN
		init := TRUE;

		dat[00] := 0;
		dat[01] := 14;
		dat[02] := 12;
		dat[03] := 9;
		dat[04] := 9;
		dat[05] := 0;
		dat[06] := 7;
		dat[07] := 7;
		dat[08] := 0;
		dat[09] := 2;
		dat[10] := 2;
		dat[11] := 3;
		dat[12] := 3;
		dat[13] := 1;
		dat[14] := 0;
		dat[15] := 0;
		dat[16] := 17;
		dat[17] := 4;
		dat[18] := 4;
		dat[19] := 3;
		dat[20] := 3;
		dat[21] := 1;
		dat[22] := 0;
		dat[23] := 0;
		dat[24] := 17;
		dat[25] := 2;
		dat[26] := 2;
		dat[27] := 3;
		dat[28] := 3;
		dat[29] := 1;
		dat[30] := 0;
		dat[31] := 0;
		dat[32] := 17;
		dat[33] := 2;
		dat[34] := 4;
		dat[35] := 3;
		dat[36] := 3;
		dat[37] := 1;
		dat[38] := 0;
		dat[39] := 0;
		dat[40] := 17;
		dat[41] := 0;
	END_IF;

	IF ACTIVATE AND act_last = FALSE THEN
		x := LIMIT(0,WW.CUR.WEATHER_ICON,41);
		WW.CUR.WEATHER_ICON := dat[x];
		FOR i := 0 TO 4 DO
			x := LIMIT(0,WW.DAY[i].WEATHER_ICON,41);
			WW.DAY[i].WEATHER_ICON := dat[x];
		END_FOR;
	END_IF;
	act_last := ACTIVATE;

END_FUNCTION_BLOCK

PROGRAM program0
	VAR
		ACTIVATE :	BOOL;
		WW :	oscat_WORLD_WEATHER_DATA;

		func_block : WORLD_WEATHER_ICON_OSCAT_Block;
	END_VAR
	func_block.ACTIVATE := ACTIVATE;
	func_block.WW := WW;

	func_block();
	WW  := func_block.WW;
END_PROGRAM

CONFIGURATION Config0
	RESOURCE Res0 ON PLC
		TASK task0(INTERVAL := T#20ms,PRIORITY := 0);
		PROGRAM instance0 WITH task0 : program0;
	END_RESOURCE
END_CONFIGURATION

(* ---- _ARRAY_ABS.ST ---- *)
TYPE
	oscat_pt_ARRAY: ARRAY [1..100] OF REAL;
END_TYPE

FUNCTION _ARRAY_ABS : BOOL
	VAR_IN_OUT
		PT : oscat_pt_ARRAY;
	END_VAR

	VAR_INPUT
		SIZE :	UINT;
	END_VAR

	VAR
		i :	INT;
		stop :	INT;
	END_VAR

	stop := LIMIT_INT(1,UINT_TO_INT(size),1000);
	FOR i := 1 TO stop DO
		pt[i] := ABS(pt[i]);
	END_FOR;

	_ARRAY_ABS := TRUE;

END_FUNCTION

PROGRAM program0
  VAR
    LocalVar0 : oscat_pt_ARRAY;
    LocalVar1 : UINT;
	LocalOUT  : BOOL;
  END_VAR

  LocalOUT := _ARRAY_ABS(LocalVar0, LocalVar1);
END_PROGRAM

CONFIGURATION Config0
  RESOURCE Res0 ON PLC
    TASK task0(INTERVAL := T#20ms,PRIORITY := 0);
    PROGRAM instance0 WITH task0 : program0;
  END_RESOURCE
END_CONFIGURATION

(* ---- _ARRAY_ADD.ST ---- *)
TYPE
	oscat_pt_ARRAY: ARRAY [1..100] OF REAL;
END_TYPE

FUNCTION _ARRAY_ADD:	BOOL
	VAR_IN_OUT
		PT :	oscat_pt_ARRAY;
	END_VAR
	VAR_INPUT
		SIZE :	UINT;
		X :	REAL;
	END_VAR
	VAR
		i :	INT;
		stop :	INT;
	END_VAR

	stop :=LIMIT_INT(1,UINT_TO_INT(size),1000);
	FOR i := 1 TO stop DO
		pt[i] := pt[i] + X;
	END_FOR;
	_ARRAY_ADD := TRUE;

END_FUNCTION

PROGRAM program0
  VAR
    LocalVar0 : oscat_pt_ARRAY;
    LocalVar1 : UINT;
	LocalVar2 : REAL;
	LocalOUT  : BOOL;
  END_VAR

  LocalOUT := _ARRAY_ADD(LocalVar0, LocalVar1, LocalVar2);
END_PROGRAM

CONFIGURATION Config0
  RESOURCE Res0 ON PLC
    TASK task0(INTERVAL := T#20ms,PRIORITY := 0);
    PROGRAM instance0 WITH task0 : program0;
  END_RESOURCE
END_CONFIGURATION

(* ---- _BYTE_TO_DINT.ST ---- *)
FUNCTION _BYTE_TO_DINT:DINT
	VAR_INPUT
		IN :	BYTE;
	END_VAR

	_BYTE_TO_DINT := USINT_TO_DINT(BYTE_TO_USINT(IN));
END_FUNCTION

PROGRAM program0
  VAR
    LocalVar0 : BYTE;
	LocalOUT  : DINT;
  END_VAR

  LocalOUT := _BYTE_TO_DINT(LocalVar0);
END_PROGRAM

CONFIGURATION Config0
  RESOURCE Res0 ON PLC
    TASK task0(INTERVAL := T#20ms,PRIORITY := 0);
    PROGRAM instance0 WITH task0 : program0;
  END_RESOURCE
END_CONFIGURATION

(* ---- _BYTE_TO_INT.ST ---- *)
FUNCTION _BYTE_TO_INT:INT
	VAR_INPUT
		IN :	BYTE;
	END_VAR

	_BYTE_TO_INT := USINT_TO_INT(BYTE_TO_USINT(IN));
END_FUNCTION

PROGRAM program0
  VAR
    LocalVar0 : BYTE;
	LocalOUT  : INT;
  END_VAR

  LocalOUT := _BYTE_TO_INT(LocalVar0);
END_PROGRAM

CONFIGURATION Config0
  RESOURCE Res0 ON PLC
    TASK task0(INTERVAL := T#20ms,PRIORITY := 0);
    PROGRAM instance0 WITH task0 : program0;
  END_RESOURCE
END_CONFIGURATION

(* ---- _BYTE_TO_REAL.ST ---- *)
FUNCTION _BYTE_TO_REAL:REAL
	VAR_INPUT
		IN :	BYTE;
	END_VAR

	_BYTE_TO_REAL := USINT_TO_REAL(BYTE_TO_USINT(IN));
END_FUNCTION

PROGRAM program0
  VAR
    LocalVar0 : BYTE;
	LocalOUT  : REAL;
  END_VAR

  LocalOUT := _BYTE_TO_REAL(LocalVar0);
END_PROGRAM

CONFIGURATION Config0
  RESOURCE Res0 ON PLC
    TASK task0(INTERVAL := T#20ms,PRIORITY := 0);
    PROGRAM instance0 WITH task0 : program0;
  END_RESOURCE
END_CONFIGURATION

(* ---- _DWORD_TO_REAL.ST ---- *)
FUNCTION _DWORD_TO_REAL:REAL
	VAR_INPUT
		IN :	DWORD;
	END_VAR

	_DWORD_TO_REAL := UDINT_TO_REAL(DWORD_TO_UDINT(IN));
END_FUNCTION

PROGRAM program0
  VAR
    LocalVar0 : DWORD;
    LocalOUT  : REAL;
  END_VAR

  LocalOUT := _DWORD_TO_REAL(LocalVar0);
END_PROGRAM

CONFIGURATION Config0
  RESOURCE Res0 ON PLC
    TASK task0(INTERVAL := T#20ms,PRIORITY := 0);
    PROGRAM instance0 WITH task0 : program0;
  END_RESOURCE
END_CONFIGURATION

(* ---- _INT_TO_UDINT.ST ---- *)
FUNCTION _INT_TO_UDINT:UDINT
	VAR_INPUT
		IN :	INT;
	END_VAR

	_INT_TO_UDINT := DINT_TO_UDINT(INT_TO_DINT(IN));
END_FUNCTION

PROGRAM program0
  VAR
    LocalVar0 : INT;
	LocalOUT  : UDINT;
  END_VAR

  LocalOUT := _INT_TO_UDINT(LocalVar0);
END_PROGRAM

CONFIGURATION Config0
  RESOURCE Res0 ON PLC
    TASK task0(INTERVAL := T#20ms,PRIORITY := 0);
    PROGRAM instance0 WITH task0 : program0;
  END_RESOURCE
END_CONFIGURATION

(* ---- _MOD_INT.ST ---- *)
FUNCTION _MOD_INT:INT
  VAR_INPUT
    IN :	INT;
    DIVISOR :	INT;
  END_VAR

  IF IN = 0 THEN
    _MOD_INT := 0;
  ELSE
    _MOD_INT := IN MOD DIVISOR;
  END_IF;
END_FUNCTION

PROGRAM program0
  VAR
    LocalVar0 : INT;
    LocalVar1 : INT;
	  LocalOUT  : INT;
  END_VAR

  LocalOUT := _MOD_INT(LocalVar0, LocalVar1);
END_PROGRAM

CONFIGURATION Config0
  RESOURCE Res0 ON PLC
    TASK task0(INTERVAL := T#20ms,PRIORITY := 0);
    PROGRAM instance0 WITH task0 : program0;
  END_RESOURCE
END_CONFIGURATION

(* ---- _REAL_TO_DINT.ST ---- *)
FUNCTION _REAL_TO_DINT:DINT
  VAR_INPUT
    X :	REAL;
  END_VAR

  IF REAL_TO_DINT(0.5) = DINT#1 THEN
    _REAL_TO_DINT := REAL_TO_DINT(x);
    RETURN;
  END_IF;

  IF X > 0.0 THEN
    _REAL_TO_DINT := REAL_TO_DINT(x+0.5);
  ELSIF X < 0.0 THEN
    _REAL_TO_DINT := REAL_TO_DINT(x-0.5);
  ELSE
    _REAL_TO_DINT := DINT#0;
  END_IF;
END_FUNCTION

PROGRAM program0
  VAR
    LocalVar0 : REAL;
	  LocalOUT  : DINT;
  END_VAR

  LocalOUT := _REAL_TO_DINT(LocalVar0);
END_PROGRAM

CONFIGURATION Config0
  RESOURCE Res0 ON PLC
    TASK task0(INTERVAL := T#20ms,PRIORITY := 0);
    PROGRAM instance0 WITH task0 : program0;
  END_RESOURCE
END_CONFIGURATION

(* ---- _REAL_TO_DWORD.ST ---- *)
FUNCTION _REAL_TO_DWORD: DWORD

  VAR_INPUT
    X :	REAL;
  END_VAR

  IF REAL_TO_DWORD(0.5) = DWORD#1 THEN
    _REAL_TO_DWORD := REAL_TO_DWORD(x);
  ELSIF X > 0.0 THEN
    _REAL_TO_DWORD := REAL_TO_DWORD(x+0.5);
  ELSIF X < 0.0 THEN
    _REAL_TO_DWORD := REAL_TO_DWORD(x-0.5);
  ELSE
    _REAL_TO_DWORD := DWORD#0;
  END_IF;
END_FUNCTION

PROGRAM program0
  VAR
    LocalVar0 : REAL;
    LocalOUT  : DWORD;
  END_VAR

  LocalOUT := _REAL_TO_DWORD(LocalVar0);
END_PROGRAM

CONFIGURATION Config0
  RESOURCE Res0 ON PLC
    TASK task0(INTERVAL := T#20ms,PRIORITY := 0);
    PROGRAM instance0 WITH task0 : program0;
  END_RESOURCE
END_CONFIGURATION

(* ---- _REAL_TO_UDINT.ST ---- *)
FUNCTION _REAL_TO_UDINT:UDINT
  VAR_INPUT
    X :	REAL;
  END_VAR

  IF REAL_TO_UDINT(0.5) = UDINT#1 THEN
    _REAL_TO_UDINT := REAL_TO_UDINT(x);
  ELSIF X > 0.0 THEN
    _REAL_TO_UDINT := REAL_TO_UDINT(x+0.5);
  ELSIF X < 0.0 THEN
    _REAL_TO_UDINT := REAL_TO_UDINT(x-0.5);
  ELSE
    _REAL_TO_UDINT := UDINT#0;
  END_IF;
END_FUNCTION

PROGRAM program0
    VAR
      LocalVar0 : REAL;
      LocalOUT  : UDINT;
    END_VAR

    LocalOUT := _REAL_TO_UDINT(LocalVar0);
END_PROGRAM

CONFIGURATION Config0
    RESOURCE Res0 ON PLC
      TASK task0(INTERVAL := T#20ms,PRIORITY := 0);
      PROGRAM instance0 WITH task0 : program0;
    END_RESOURCE
END_CONFIGURATION

(* ---- _WORD_TO_DINT.ST ---- *)
FUNCTION _WORD_TO_DINT:DINT
	VAR_INPUT
		IN :	WORD;
	END_VAR
	_WORD_TO_DINT := UINT_TO_DINT(WORD_TO_UINT(IN));
END_FUNCTION
PROGRAM program0
  VAR
    LocalVar0 : WORD;
    LocalOUT  : DINT;
  END_VAR

  LocalOUT := _WORD_TO_DINT(LocalVar0);
END_PROGRAM

CONFIGURATION Config0
  RESOURCE Res0 ON PLC
    TASK task0(INTERVAL := T#20ms,PRIORITY := 0);
    PROGRAM instance0 WITH task0 : program0;
  END_RESOURCE
END_CONFIGURATION

(* ---- _WORD_TO_REAL.ST ---- *)
FUNCTION _WORD_TO_REAL:REAL
	VAR_INPUT
		IN :	WORD;
	END_VAR
	_WORD_TO_REAL := UINT_TO_REAL(WORD_TO_UINT(IN));
END_FUNCTION

PROGRAM program0
  VAR
    LocalVar0 : WORD;
    LocalOUT  : REAL;
  END_VAR

  LocalOUT := _WORD_TO_REAL(LocalVar0);
END_PROGRAM

CONFIGURATION Config0
  RESOURCE Res0 ON PLC
    TASK task0(INTERVAL := T#20ms,PRIORITY := 0);
    PROGRAM instance0 WITH task0 : program0;
  END_RESOURCE
END_CONFIGURATION

(* ---- ACOSH.ST ---- *)
FUNCTION ACOSH:REAL
	VAR_INPUT
		X :	REAL;
	END_VAR
	ACOSH := LN(SQRT(X * X - 1.0) + X);

END_FUNCTION

PROGRAM program0
  VAR
    LocalVar0 : REAL;
    LocalOUT  : REAL;
  END_VAR

  LocalOUT := ACOSH(LocalVar0);
END_PROGRAM

CONFIGURATION Config0
  RESOURCE Res0 ON PLC
    TASK task0(INTERVAL := T#20ms,PRIORITY := 0);
    PROGRAM instance0 WITH task0 : program0;
  END_RESOURCE
END_CONFIGURATION

(* ---- ACOTH.ST ---- *)
FUNCTION ACOTH:REAL
	VAR_INPUT
		X :	REAL;
	END_VAR

	ACOTH := LN((x+1.0)/(x-1.0))*0.5;

END_FUNCTION

PROGRAM program0
  VAR
    LocalVar0 : REAL;
    LocalOUT  : REAL;
  END_VAR

  LocalOUT := ACOTH(LocalVar0);
END_PROGRAM

CONFIGURATION Config0
  RESOURCE Res0 ON PLC
    TASK task0(INTERVAL := T#20ms,PRIORITY := 0);
    PROGRAM instance0 WITH task0 : program0;
  END_RESOURCE
END_CONFIGURATION

(* ---- AGDF.ST ---- *)
FUNCTION AGDF:REAL
	VAR_INPUT
		X :	REAL;
	END_VAR

	AGDF := LN((1.0 + SIN(X)) / COS(X));
END_FUNCTION

PROGRAM program0
  VAR
    LocalVar0 : REAL;
    LocalOUT  : REAL;
  END_VAR

  LocalOUT := AGDF(LocalVar0);
END_PROGRAM

CONFIGURATION Config0
  RESOURCE Res0 ON PLC
    TASK task0(INTERVAL := T#20ms,PRIORITY := 0);
    PROGRAM instance0 WITH task0 : program0;
  END_RESOURCE
END_CONFIGURATION

(* ---- AIN.ST ---- *)
FUNCTION _BYTE_TO_INT:INT
	VAR_INPUT
		IN :	BYTE;
	END_VAR

	_BYTE_TO_INT := USINT_TO_INT(BYTE_TO_USINT(IN));
END_FUNCTION

FUNCTION _DWORD_TO_REAL:REAL
	VAR_INPUT
		IN :	DWORD;
	END_VAR

	_DWORD_TO_REAL := UDINT_TO_REAL(DWORD_TO_UDINT(IN));
END_FUNCTION

FUNCTION BIT_OF_DWORD:BOOL
	VAR_INPUT
		IN :	DWORD;
		N :	INT;
	END_VAR
	BIT_OF_DWORD := (SHR(in,n) AND DWORD#1) > DWORD#0;
END_FUNCTION

FUNCTION AIN:REAL
	VAR_INPUT
		IN :	DWORD;
		BITS :	BYTE;
		SIGN :	BYTE;
		LOW :	REAL;
		HIGH :	REAL;
	END_VAR

	VAR
		temp1 :	DWORD;
		temp2 :	DWORD;
		sx :	BOOL;
	END_VAR

	IF sign < BYTE#32 THEN
		temp1 := SHR(in, _BYTE_TO_INT(sign));
		sx := BIT_OF_DWORD(temp1,0); (* temp1.X0 *)
	ELSE
		sx := FALSE;
	END_IF;
	temp1 := SHR(DWORD#16#FFFFFFFF,32 - _BYTE_TO_INT(bits));
	temp2 := in AND temp1;
	AIN := (high - low)* _DWORD_TO_REAL(temp2) / _DWORD_TO_REAL(temp1) + low;
	IF sx THEN AIN := -AIN; END_IF;
END_FUNCTION

PROGRAM program0
  VAR
    LocalVar0 : DWORD;
	LocalVar1 : BYTE;
	LocalVar2 : BYTE;
	LocalVar3 : REAL;
	LocalVar4 : REAL;
    LocalOUT  : REAL;
  END_VAR

  LocalOUT := AIN(LocalVar0, LocalVar1, LocalVar2, LocalVar3, LocalVar4);
END_PROGRAM

CONFIGURATION Config0
  RESOURCE Res0 ON PLC
    TASK task0(INTERVAL := T#20ms,PRIORITY := 0);
    PROGRAM instance0 WITH task0 : program0;
  END_RESOURCE
END_CONFIGURATION

(* ---- AIR_DENSITY.ST ---- *)
FUNCTION SDD:REAL

	VAR_INPUT
		T :	REAL;
		ICE :	BOOL;
	END_VAR

	IF ice THEN
		SDD := 611.153 * EXP(22.4433 * T / (272.186 + T));
	ELSE
		SDD := 611.213 * EXP(17.5043 * T / (241.2 + T));
	END_IF;

END_FUNCTION

FUNCTION AIR_DENSITY:REAL

	VAR_INPUT
		T :	REAL;
		P :	REAL;
		RH :	REAL;
	END_VAR

	AIR_DENSITY := 101325.0 * (1.0 - RH * SDD(T, TRUE) * 3.773319E-3 / P) / (287.05 * ( T - -273.15));

END_FUNCTION

PROGRAM program0
  VAR
    T :	REAL;
	P :	REAL;
	RH :	REAL;
    CEIL5_OUT : REAL;
  END_VAR

  CEIL5_OUT := AIR_DENSITY(T, P, RH);
END_PROGRAM

CONFIGURATION Config0

  RESOURCE Res0 ON PLC
    TASK task0(INTERVAL := T#20ms,PRIORITY := 0);
    PROGRAM instance0 WITH task0 : program0;
  END_RESOURCE
END_CONFIGURATION

(* ---- AIR_ENTHALPY.ST ---- *)
FUNCTION SDD:REAL

	VAR_INPUT
		T :	REAL;
		ICE :	BOOL;
	END_VAR

	IF ice THEN
		SDD := 611.153 * EXP(22.4433 * T / (272.186 + T));
	ELSE
		SDD := 611.213 * EXP(17.5043 * T / (241.2 + T));
	END_IF;

END_FUNCTION

FUNCTION DEW_CON:REAL

	VAR_INPUT
		RH :	REAL;
		T :	REAL;
	END_VAR

	IF RH > 0.0 AND T > -50.0 THEN
		DEW_CON := 2.166824303E-2 * RH * SDD(T,FALSE)  / (T - -273.15);
	ELSE
		DEW_CON := 0.0;
	END_IF;

END_FUNCTION

FUNCTION AIR_ENTHALPY:REAL

	VAR_INPUT
		T :	REAL;
		RH :	REAL;
	END_VAR

	Air_enthalpy := 1.00482 * T + (1.86 * T + 2500.78) * dew_con(RH,T);

END_FUNCTION

PROGRAM program0
  VAR
    T :	REAL;
	RH :	REAL;
    CEIL5_OUT : REAL;
  END_VAR

  CEIL5_OUT := AIR_ENTHALPY(T, RH);
END_PROGRAM

CONFIGURATION Config0

  RESOURCE Res0 ON PLC
    TASK task0(INTERVAL := T#20ms,PRIORITY := 0);
    PROGRAM instance0 WITH task0 : program0;
  END_RESOURCE
END_CONFIGURATION

(* ---- AOUT.ST ---- *)
FUNCTION _DWORD_TO_REAL:REAL
	VAR_INPUT
		IN :	DWORD;
	END_VAR

	_DWORD_TO_REAL := UDINT_TO_REAL(DWORD_TO_UDINT(IN));
END_FUNCTION

FUNCTION SIGN_R : BOOL
  VAR_INPUT
    IN : REAL;
  END_VAR
  SIGN_R := in < 0.0;
END_FUNCTION

FUNCTION _REAL_TO_DWORD: DWORD

  VAR_INPUT
    X :	REAL;
  END_VAR

  IF REAL_TO_DWORD(0.5) = DWORD#1 THEN
    _REAL_TO_DWORD := REAL_TO_DWORD(x);
  ELSIF X > 0.0 THEN
    _REAL_TO_DWORD := REAL_TO_DWORD(x+0.5);
  ELSIF X < 0.0 THEN
    _REAL_TO_DWORD := REAL_TO_DWORD(x-0.5);
  ELSE
    _REAL_TO_DWORD := DWORD#0;
  END_IF;
END_FUNCTION

FUNCTION _BYTE_TO_INT:INT
	VAR_INPUT
		IN :	BYTE;
	END_VAR

	_BYTE_TO_INT := USINT_TO_INT(BYTE_TO_USINT(IN));
END_FUNCTION

FUNCTION AOUT:DWORD
	VAR_INPUT
		IN :	REAL;
		BITS :	BYTE;
		SIGN :	BYTE;
		LOW :	REAL;
		HIGH :	REAL;
	END_VAR

	VAR
		in2 :	REAL;
		sx :	BOOL;
	END_VAR

	IF sign < BYTE#32 THEN
		sx := sign_R(in);
		in2 := ABS(in);
	ELSE
		in2 := in;
	END_IF;

	in2 := LIMIT(low, in2, high);

	Aout := _REAL_TO_DWORD((in2 - low) / (high - low) * (_DWORD_TO_REAL(SHL(DWORD#2#1,_BYTE_TO_INT(bits))) - 1.0)   );
	IF sx THEN Aout := SHL(DWORD#2#1,_BYTE_TO_INT(sign)) OR Aout; END_IF;

END_FUNCTION

PROGRAM program0
  VAR
    LocalVar0 : REAL;
	LocalVar1 : BYTE;
	LocalVar2 : BYTE;
	LocalVar3 : REAL;
	LocalVar4 : REAL;
	LocalOUT  : DWORD;
  END_VAR
  	LocalOUT := AOUT(LocalVar0, LocalVar1, LocalVar2, LocalVar3,LocalVar4);
END_PROGRAM

CONFIGURATION Config0
  RESOURCE Res0 ON PLC
    TASK task0(INTERVAL := T#20ms,PRIORITY := 0);
    PROGRAM instance0 WITH task0 : program0;
  END_RESOURCE
END_CONFIGURATION

(* ---- AOUT1.ST ---- *)
FUNCTION SIGN_R : BOOL
  VAR_INPUT
    IN : REAL;
  END_VAR

  SIGN_R := in < 0.0;
END_FUNCTION

FUNCTION _REAL_TO_DWORD: DWORD

  VAR_INPUT
    X :	REAL;
  END_VAR

  IF REAL_TO_DWORD(0.5) = DWORD#1 THEN
    _REAL_TO_DWORD := REAL_TO_DWORD(x);
  ELSIF X > 0.0 THEN
    _REAL_TO_DWORD := REAL_TO_DWORD(x+0.5);
  ELSIF X < 0.0 THEN
    _REAL_TO_DWORD := REAL_TO_DWORD(x-0.5);
  ELSE
    _REAL_TO_DWORD := DWORD#0;
  END_IF;
END_FUNCTION

FUNCTION AOUT1:DWORD

	VAR_INPUT
		IN :	REAL;
		BIT_0 :	INT;
		BIT_N :	INT;
		SIGN :	INT;
		LOW :	REAL;
		HIGH :	REAL;
	END_VAR

	VAR
		in2 :	REAL;
		sx :	BOOL;
	END_VAR

	IF sign < 32 THEN
		sx := sign_R(in);
		in2 := ABS(in);
	ELSE
		sx := FALSE;
		in2 := in;
	END_IF;

	in2 := LIMIT_REAL(low, in2, high);

	AOUT1 :=  SHL(_REAL_TO_DWORD((in2 - low) / (high - low) * UDINT_TO_REAL(DWORD_TO_UDINT(SHL(DWORD#2#1,bit_n - Bit_0 + 1)) - UDINT#1)),Bit_0);

	IF sx THEN AOUT1 := SHL(DWORD#2#1,sign) OR AOUT1; END_IF;

END_FUNCTION

PROGRAM program0
  VAR
    LocalVar0 : REAL;
	LocalVar1 : INT;
	LocalVar21 : INT;
	LocalVar2 : INT;
	LocalVar3 : REAL;
	LocalVar4 : REAL;
	LocalOUT  : DWORD;
  END_VAR
  	LocalOUT := AOUT1(LocalVar0, LocalVar1,LocalVar21, LocalVar2, LocalVar3,LocalVar4);
END_PROGRAM

CONFIGURATION Config0
  RESOURCE Res0 ON PLC
    TASK task0(INTERVAL := T#20ms,PRIORITY := 0);
    PROGRAM instance0 WITH task0 : program0;
  END_RESOURCE
END_CONFIGURATION

(* ---- ASINH.ST ---- *)
FUNCTION ASINH:REAL
	VAR_INPUT
		X :	REAL;
	END_VAR

	ASINH := LN(SQRT(X * X + 1.0)+X);
END_FUNCTION

PROGRAM program0
  VAR
    LocalVar0 : REAL;
    LocalOUT  : REAL;
  END_VAR

  LocalOUT := ASINH(LocalVar0);
END_PROGRAM

CONFIGURATION Config0
  RESOURCE Res0 ON PLC
    TASK task0(INTERVAL := T#20ms,PRIORITY := 0);
    PROGRAM instance0 WITH task0 : program0;
  END_RESOURCE
END_CONFIGURATION

(* ---- ATAN2.ST ---- *)
FUNCTION ATAN2:REAL
	VAR_INPUT
		X :	REAL;
		Y :	REAL;
	END_VAR

	IF X > 0.0 THEN
		ATAN2 := ATAN(Y/X);
	ELSIF X < 0.0 THEN
		IF Y >= 0.0 THEN
			ATAN2 := ATAN(Y/X) + 3.14159265358979323846264338327950288;
		ELSE
			ATAN2 := ATAN(Y/X) - 3.14159265358979323846264338327950288;
		END_IF;
	ELSIF Y > 0.0 THEN
		ATAN2 := 1.5707963267948965580;
	ELSIF Y < 0.0 THEN
		ATAN2 := -1.5707963267948965580;
	ELSE
		ATAN2 := 0.0;
	END_IF;

END_FUNCTION

PROGRAM program0
  VAR
    LocalVar0 : REAL;
	LocalVar1 : REAL;
    LocalOUT  : REAL;
  END_VAR

  LocalOUT := ATAN2(LocalVar0, LocalVar1);
END_PROGRAM

CONFIGURATION Config0
  RESOURCE Res0 ON PLC
    TASK task0(INTERVAL := T#20ms,PRIORITY := 0);
    PROGRAM instance0 WITH task0 : program0;
  END_RESOURCE
END_CONFIGURATION

(* ---- ATANH.ST ---- *)
FUNCTION ATANH:REAL
	VAR_INPUT
		X :	REAL;
	END_VAR

	ATANH := LN((1.0 + x)/(1.0 - x)) * 0.5;

END_FUNCTION

PROGRAM program0
  VAR
    LocalVar0 : REAL;
    LocalOUT  : REAL;
  END_VAR

  LocalOUT := ATANH(LocalVar0);
END_PROGRAM

CONFIGURATION Config0
  RESOURCE Res0 ON PLC
    TASK task0(INTERVAL := T#20ms,PRIORITY := 0);
    PROGRAM instance0 WITH task0 : program0;
  END_RESOURCE
END_CONFIGURATION

(* ---- BAND_B.ST ---- *)
FUNCTION BAND_B:BYTE
	VAR_INPUT
		X :	BYTE;
		B :	BYTE;
	END_VAR

	IF X < B THEN
		BAND_B := BYTE#0;
	ELSIF X > USINT_TO_BYTE(USINT#255 - BYTE_TO_USINT(B)) THEN
		BAND_B := BYTE#255;
	ELSE
		BAND_B := X;
	END_IF;
END_FUNCTION
PROGRAM program0
  VAR
    LocalVar0 : BYTE;
	LocalVar1 : BYTE;
    LocalOUT  : BYTE;
  END_VAR

  LocalOUT := BAND_B(LocalVar0, LocalVar1);
END_PROGRAM

CONFIGURATION Config0
  RESOURCE Res0 ON PLC
    TASK task0(INTERVAL := T#20ms,PRIORITY := 0);
    PROGRAM instance0 WITH task0 : program0;
  END_RESOURCE
END_CONFIGURATION

(* ---- BCDC_TO_INT.ST ---- *)
FUNCTION _BYTE_TO_INT:INT
	VAR_INPUT
		IN :	BYTE;
	END_VAR

	_BYTE_TO_INT := USINT_TO_INT(BYTE_TO_USINT(IN));

END_FUNCTION

FUNCTION BCDC_TO_INT:INT
	VAR_INPUT
		IN :	BYTE;
	END_VAR

	BCDC_TO_INT := _BYTE_TO_INT(in AND BYTE#16#0F) + (_BYTE_TO_INT(SHR(in,4)) * 10);
END_FUNCTION

PROGRAM program0
  VAR
    LocalVar0 : BYTE;
    LocalOUT  : INT;
  END_VAR

  LocalOUT := BCDC_TO_INT(LocalVar0);
END_PROGRAM

CONFIGURATION Config0
  RESOURCE Res0 ON PLC
    TASK task0(INTERVAL := T#20ms,PRIORITY := 0);
    PROGRAM instance0 WITH task0 : program0;
  END_RESOURCE
END_CONFIGURATION

(* ---- BETA.ST ---- *)
FUNCTION GAMMA:REAL
	VAR_INPUT
		X :	REAL;
	END_VAR

	IF x > 0.0 THEN
		GAMMA := SQRT(6.28318530717958647692528676655900576 / X) * EXPT(0.367879441171442 * (x + 1.0 / (12.0 * x - 0.1 / X)), X);
	END_IF;
END_FUNCTION

FUNCTION BETA:REAL

	VAR_INPUT
		X :	REAL;
		Y :	REAL;
	END_VAR

	BETA := GAMMA(X)*GAMMA(Y) / GAMMA(x+y);

END_FUNCTION

PROGRAM program0
  VAR
    LocalVar0 : REAL;
	LocalVar1 : REAL;
    LocalOUT  : REAL;
  END_VAR

  LocalOUT := BETA(LocalVar0, LocalVar1);
END_PROGRAM

CONFIGURATION Config0
  RESOURCE Res0 ON PLC
    TASK task0(INTERVAL := T#20ms,PRIORITY := 0);
    PROGRAM instance0 WITH task0 : program0;
  END_RESOURCE
END_CONFIGURATION

(* ---- BFT_TO_MS.ST ---- *)
FUNCTION BFT_TO_MS:REAL
	VAR_INPUT
		BFT :	INT;
	END_VAR

	BFT_TO_MS := EXPT(INT_TO_REAL(BFT), 1.5) * 0.836;

END_FUNCTION

PROGRAM program0
  VAR
    LocalVar0 : INT;
    LocalOUT  : REAL;
  END_VAR

  LocalOUT := BFT_TO_MS(LocalVar0);
END_PROGRAM

CONFIGURATION Config0
  RESOURCE Res0 ON PLC
    TASK task0(INTERVAL := T#20ms,PRIORITY := 0);
    PROGRAM instance0 WITH task0 : program0;
  END_RESOURCE
END_CONFIGURATION

(* ---- BINOM.ST ---- *)
FUNCTION BINOM:INT
	VAR_INPUT
		N :	INT;
		K :	INT;
	END_VAR

	VAR
		i :	INT;
		N2 :	INT;
		K2 :	INT;
	END_VAR

	K2 := K;
	N2 := N;
	IF 2 * K2 > N2 THEN
		K2 := N2 - K2;
	END_IF;
	IF K2 > N2 THEN
		RETURN;
	ELSIF K2 = 0 OR K2 = N2 THEN
		BINOM := 1;
	ELSIF K2 = 1 THEN
		BINOM := N2;
	ELSE
		BINOM := N2;
		N2 := N2 + 1;
		FOR i := 2 TO K2 DO
			BINOM := BINOM * (N2 - i) / i;
		END_FOR;
	END_IF;
END_FUNCTION

PROGRAM program0
  VAR
    LocalVar0 : INT;
	LocalVar1 : INT;
    LocalOUT  : INT;
  END_VAR

  LocalOUT := BINOM(LocalVar0, LocalVar1);
END_PROGRAM

CONFIGURATION Config0
  RESOURCE Res0 ON PLC
    TASK task0(INTERVAL := T#20ms,PRIORITY := 0);
    PROGRAM instance0 WITH task0 : program0;
  END_RESOURCE
END_CONFIGURATION

(* ---- BIT_COUNT.ST ---- *)
FUNCTION BIT_COUNT:INT

	VAR_INPUT
		IN :	DWORD;
	END_VAR

	VAR
		in_temp :	DWORD;
	END_VAR

	in_temp := IN;
	WHILE in_temp > DWORD#0 DO
		IF (in_temp AND DWORD#16#00000001) > DWORD#0 THEN Bit_Count := Bit_Count +1; END_IF;
		in_temp := SHR(in_temp,1);
	END_WHILE;

END_FUNCTION

PROGRAM program0
  VAR
    LocalVar0 : DWORD;
    LocalOUT  : INT;
  END_VAR

  LocalOUT := BIT_COUNT(LocalVar0);
END_PROGRAM

CONFIGURATION Config0
  RESOURCE Res0 ON PLC
    TASK task0(INTERVAL := T#20ms,PRIORITY := 0);
    PROGRAM instance0 WITH task0 : program0;
  END_RESOURCE
END_CONFIGURATION

(* ---- BIT_LOAD_B.ST ---- *)
FUNCTION BIT_LOAD_B:BYTE
	VAR_INPUT
		IN :	BYTE;
		VAL :	BOOL;
		POS :	INT;
	END_VAR

	IF VAL THEN
		BIT_LOAD_B := in OR SHL(BYTE#1,pos);
	ELSE
		BIT_LOAD_B := in AND (NOT SHL(BYTE#1,pos));
	END_IF;
END_FUNCTION

PROGRAM program0
  VAR
    LocalVar0 : BYTE;
	LocalVar1 : BOOL;
	LocalVar2 : INT;
    LocalOUT  : BYTE;
  END_VAR

  LocalOUT := BIT_LOAD_B(LocalVar0, LocalVar1, LocalVar2);
END_PROGRAM

CONFIGURATION Config0
  RESOURCE Res0 ON PLC
    TASK task0(INTERVAL := T#20ms,PRIORITY := 0);
    PROGRAM instance0 WITH task0 : program0;
  END_RESOURCE
END_CONFIGURATION

(* ---- BIT_LOAD_B2.ST ---- *)
FUNCTION BIT_LOAD_B2:BYTE
	VAR_INPUT
		I :	BYTE;
		D :	BOOL;
		P :	INT;
		N :	INT;
	END_VAR

	IF D THEN
		BIT_LOAD_B2 := ROL(SHR(BYTE#255, 8 - N) OR ROR(I, P), P);
	ELSE
		BIT_LOAD_B2 := ROL(SHL(BYTE#255, N) AND ROR(I, P), P);
	END_IF;
END_FUNCTION

PROGRAM program0
  VAR
    LocalVar0 : BYTE;
	LocalVar1 : BOOL;
	LocalVar2 : INT;
	LocalVar3 : INT;
    LocalOUT  : BYTE;
  END_VAR

  LocalOUT := BIT_LOAD_B2(LocalVar0, LocalVar1, LocalVar2, LocalVar3);
END_PROGRAM

CONFIGURATION Config0
  RESOURCE Res0 ON PLC
    TASK task0(INTERVAL := T#20ms,PRIORITY := 0);
    PROGRAM instance0 WITH task0 : program0;
  END_RESOURCE
END_CONFIGURATION

(* ---- BIT_LOAD_DW.ST ---- *)
FUNCTION BIT_LOAD_DW:DWORD

	VAR_INPUT
		IN :	DWORD;
		VAL :	BOOL;
		POS :	INT;
	END_VAR

	IF val THEN
		BIT_LOAD_DW := in OR SHL(DWORD#1,pos);
	ELSE
		BIT_LOAD_DW := in AND (NOT SHL(DWORD#1,pos));
	END_IF;

END_FUNCTION

PROGRAM program0
  VAR
    LocalVar0 : DWORD;
	LocalVar1 : BOOL;
	LocalVar2 : INT;
    LocalOUT  : DWORD;
  END_VAR

  LocalOUT := BIT_LOAD_DW(LocalVar0, LocalVar1, LocalVar2);
END_PROGRAM

CONFIGURATION Config0
  RESOURCE Res0 ON PLC
    TASK task0(INTERVAL := T#20ms,PRIORITY := 0);
    PROGRAM instance0 WITH task0 : program0;
  END_RESOURCE
END_CONFIGURATION

(* ---- BIT_LOAD_DW2.ST ---- *)
FUNCTION BIT_LOAD_DW2:DWORD
	VAR_INPUT
		I :	DWORD;
		D :	BOOL;
		P :	INT;
		N :	INT;
	END_VAR

	IF D THEN
		BIT_LOAD_DW2 := ROL(SHR(DWORD#16#FFFFFFFF, 32 - N) OR ROR(I, P), P);
	ELSE
		BIT_LOAD_DW2 := ROL(SHL(DWORD#16#FFFFFFFF, N) AND ROR(I, P), P);
	END_IF;

END_FUNCTION

PROGRAM program0
  VAR
    LocalVar0 : DWORD;
	LocalVar1 : BOOL;
	LocalVar2 : INT;
	LocalVar3 : INT;
    LocalOUT  : DWORD;
  END_VAR

  LocalOUT := BIT_LOAD_DW2(LocalVar0, LocalVar1, LocalVar2, LocalVar3);
END_PROGRAM

CONFIGURATION Config0
  RESOURCE Res0 ON PLC
    TASK task0(INTERVAL := T#20ms,PRIORITY := 0);
    PROGRAM instance0 WITH task0 : program0;
  END_RESOURCE
END_CONFIGURATION

(* ---- BIT_LOAD_W.ST ---- *)
FUNCTION BIT_LOAD_W:WORD
	VAR_INPUT
		IN :	WORD;
		VAL :	BOOL;
		POS :	INT;
	END_VAR

	IF VAL THEN
		BIT_LOAD_W := in OR SHL(WORD#1,pos);
	ELSE
		BIT_LOAD_W := in AND (NOT SHL(WORD#1,pos));
	END_IF;
END_FUNCTION

PROGRAM program0
  VAR
    LocalVar0 : WORD;
	LocalVar1 : BOOL;
	LocalVar2 : INT;
    LocalOUT  : WORD;
  END_VAR

  LocalOUT := BIT_LOAD_W(LocalVar0, LocalVar1, LocalVar2);
END_PROGRAM

CONFIGURATION Config0
  RESOURCE Res0 ON PLC
    TASK task0(INTERVAL := T#20ms,PRIORITY := 0);
    PROGRAM instance0 WITH task0 : program0;
  END_RESOURCE
END_CONFIGURATION

(* ---- BIT_LOAD_W2.ST ---- *)
FUNCTION BIT_LOAD_W2:WORD
	VAR_INPUT
		I :	WORD;
		D :	BOOL;
		P :	INT;
		N :	INT;
	END_VAR

	IF D THEN
		BIT_LOAD_W2 := ROL(SHR(WORD#16#FFFF, 16 - N) OR ROR(I, P), P);
	ELSE
		BIT_LOAD_W2 := ROL(SHL(WORD#16#FFFF, N) AND ROR(I, P), P);
	END_IF;
END_FUNCTION

PROGRAM program0
  VAR
    LocalVar0 : WORD;
	LocalVar1 : BOOL;
	LocalVar2 : INT;
	LocalVar3 : INT;
    LocalOUT  : WORD;
  END_VAR

  LocalOUT := BIT_LOAD_W2(LocalVar0, LocalVar1, LocalVar2, LocalVar3);
END_PROGRAM

CONFIGURATION Config0
  RESOURCE Res0 ON PLC
    TASK task0(INTERVAL := T#20ms,PRIORITY := 0);
    PROGRAM instance0 WITH task0 : program0;
  END_RESOURCE
END_CONFIGURATION

(* ---- BIT_OF_DWORD.ST ---- *)
FUNCTION BIT_OF_DWORD : BOOL
  VAR_INPUT
    IN : DWORD;
    N : INT;
  END_VAR

  BIT_OF_DWORD := (SHR(in,N) AND 16#00000001) > 0;
END_FUNCTION

PROGRAM program0
  VAR
    LocalVar0 : DWORD;
    LocalVar2 : INT;
    LocalVar1 : BOOL;
    CEIL5_OUT : BOOL;
  END_VAR

  CEIL5_OUT := BIT_OF_DWORD(LocalVar0, LocalVar2);
  LocalVar1 := CEIL5_OUT;
END_PROGRAM

CONFIGURATION Config0

  RESOURCE Res0 ON PLC
    TASK task0(INTERVAL := T#20ms,PRIORITY := 0);
    PROGRAM instance0 WITH task0 : program0;
  END_RESOURCE
END_CONFIGURATION

(* ---- BIT_TOGGLE_B.ST ---- *)
FUNCTION BIT_TOGGLE_B:BYTE
	VAR_INPUT
		IN :	BYTE;
		POS :	INT;
	END_VAR

	BIT_TOGGLE_B := SHL(BYTE#1, POS) XOR IN;
END_FUNCTION

PROGRAM program0
  VAR
    LocalVar0 : BYTE;
    LocalVar1 : INT;
    CEIL5_OUT : BYTE;
  END_VAR

  CEIL5_OUT := BIT_TOGGLE_B(LocalVar0, LocalVar1);
END_PROGRAM

CONFIGURATION Config0

  RESOURCE Res0 ON PLC
    TASK task0(INTERVAL := T#20ms,PRIORITY := 0);
    PROGRAM instance0 WITH task0 : program0;
  END_RESOURCE
END_CONFIGURATION

(* ---- BIT_TOGGLE_DW.ST ---- *)
FUNCTION BIT_TOGGLE_DW:DWORD
	VAR_INPUT
		IN :	DWORD;
		POS :	INT;
	END_VAR

	BIT_TOGGLE_DW := SHL(DWORD#1, POS) XOR IN;

END_FUNCTION

PROGRAM program0
  VAR
    LocalVar0 : DWORD;
    LocalVar1 : INT;
    CEIL5_OUT : DWORD;
  END_VAR

  CEIL5_OUT := BIT_TOGGLE_DW(LocalVar0, LocalVar1);
END_PROGRAM

CONFIGURATION Config0

  RESOURCE Res0 ON PLC
    TASK task0(INTERVAL := T#20ms,PRIORITY := 0);
    PROGRAM instance0 WITH task0 : program0;
  END_RESOURCE
END_CONFIGURATION

(* ---- BIT_TOGGLE_W.ST ---- *)
FUNCTION BIT_TOGGLE_W:WORD
	VAR_INPUT
		IN :	WORD;
		POS :	INT;
	END_VAR

	BIT_TOGGLE_W := SHL(WORD#1, POS) XOR IN;
END_FUNCTION

PROGRAM program0
  VAR
    LocalVar0 : WORD;
    LocalVar1 : INT;
    CEIL5_OUT : WORD;
  END_VAR

  CEIL5_OUT := BIT_TOGGLE_W(LocalVar0, LocalVar1);
END_PROGRAM

CONFIGURATION Config0

  RESOURCE Res0 ON PLC
    TASK task0(INTERVAL := T#20ms,PRIORITY := 0);
    PROGRAM instance0 WITH task0 : program0;
  END_RESOURCE
END_CONFIGURATION

(* ---- BUILDING_VERSION.ST ---- *)
FUNCTION _INT_TO_UDINT:UDINT
	VAR_INPUT
		IN :	INT;
	END_VAR

	_INT_TO_UDINT := DINT_TO_UDINT(INT_TO_DINT(IN));
END_FUNCTION

FUNCTION SET_DATE:UDINT

	VAR_INPUT
		YEAR :	INT;
		MONTH :	INT;
		DAY :	INT;
	END_VAR

	VAR
		count :	INT;
	END_VAR

	IF month > 2 THEN
		count := (month - 1) * 30;
		IF month > 7 THEN
			count := count + DWORD_TO_INT(SHR(DINT_TO_DWORD(INT_TO_DINT(month) - INT_TO_DINT(3)),1));
		ELSE
			count := count + DWORD_TO_INT(SHR(DINT_TO_DWORD(INT_TO_DINT(month) - INT_TO_DINT(4)),1));
		END_IF;
		IF SHL(INT_TO_WORD(year),14) = WORD#0 THEN
			count := count + 1;
		END_IF;
	ELSE
		count := (month - 1) * 31;
	END_IF;
	SET_DATE := (_INT_TO_UDINT(count + day - 1) + DWORD_TO_UDINT(SHR(UDINT_TO_DWORD(_INT_TO_UDINT(year) * UDINT#1461 - UDINT#2878169), 2))) * UDINT#86400;

END_FUNCTION

FUNCTION BUILDING_VERSION:DWORD

	VAR_INPUT
		IN :	BOOL;
	END_VAR

	IF in THEN
		BUILDING_VERSION := UDINT_TO_DWORD(set_Date(2011,02,03));
	ELSE
		BUILDING_VERSION := DWORD#100;
	END_IF;

END_FUNCTION

PROGRAM program0
	VAR
		IN :	BOOL;
		CEIL5_OUT : DWORD;
	END_VAR

  	CEIL5_OUT := BUILDING_VERSION(IN);
END_PROGRAM

CONFIGURATION Config0

  RESOURCE Res0 ON PLC
    TASK task0(INTERVAL := T#20ms,PRIORITY := 0);
    PROGRAM instance0 WITH task0 : program0;
  END_RESOURCE
END_CONFIGURATION

(* ---- BYTE_OF_BIT.ST ---- *)
FUNCTION BYTE_OF_BIT:BYTE
	VAR_INPUT
		B0 :	BOOL;
		B1 :	BOOL;
		B2 :	BOOL;
		B3 :	BOOL;
		B4 :	BOOL;
		B5 :	BOOL;
		B6 :	BOOL;
		B7 :	BOOL;
	END_VAR
	Byte_of_bit := SHL(SHL(SHL(SHL(SHL(SHL(SHL(BOOL_TO_BYTE(B7),1) OR BOOL_TO_BYTE(B6),1)
	OR BOOL_TO_BYTE(B5),1) OR BOOL_TO_BYTE(B4),1) OR BOOL_TO_BYTE(B3),1) OR BOOL_TO_BYTE(B2),1)
	OR BOOL_TO_BYTE(B1),1) OR BOOL_TO_BYTE(B0);
END_FUNCTION

PROGRAM program0
  VAR
	B0 :	BOOL;
	B1 :	BOOL;
	B2 :	BOOL;
	B3 :	BOOL;
	B4 :	BOOL;
	B5 :	BOOL;
	B6 :	BOOL;
	B7 :	BOOL;
    LocalOUT  : BYTE;
  END_VAR

  LocalOUT := BYTE_OF_BIT(B0, B1, B2, B3, B4, B5, B6, B7);
END_PROGRAM

CONFIGURATION Config0
  RESOURCE Res0 ON PLC
    TASK task0(INTERVAL := T#20ms,PRIORITY := 0);
    PROGRAM instance0 WITH task0 : program0;
  END_RESOURCE
END_CONFIGURATION

(* ---- BYTE_OF_DWORD.ST ---- *)
FUNCTION _BYTE_TO_INT:INT
	VAR_INPUT
		IN :	BYTE;
	END_VAR

	_BYTE_TO_INT := USINT_TO_INT(BYTE_TO_USINT(IN));
END_FUNCTION

FUNCTION BYTE_OF_DWORD:BYTE
	VAR_INPUT
		IN :	DWORD;
		N :	BYTE;
	END_VAR
	BYTE_OF_DWORD := DWORD_TO_BYTE(SHR(in,_BYTE_TO_INT(SHL(n,3))));
END_FUNCTION

PROGRAM program0
  VAR
    LocalVar0 : DWORD;
	  LocalVar1 : BYTE;
    LocalOUT  : BYTE;
  END_VAR

  LocalOUT := BYTE_OF_DWORD(LocalVar0, LocalVar1);
END_PROGRAM

CONFIGURATION Config0
  RESOURCE Res0 ON PLC
    TASK task0(INTERVAL := T#20ms,PRIORITY := 0);
    PROGRAM instance0 WITH task0 : program0;
  END_RESOURCE
END_CONFIGURATION

(* ---- BYTE_TO_GRAY.ST ---- *)
FUNCTION BYTE_TO_GRAY:BYTE
	VAR_INPUT
		IN :	BYTE;
	END_VAR

	BYTE_TO_GRAY := IN XOR SHR(IN,1);
END_FUNCTION

PROGRAM program0
  VAR
    LocalVar0 : BYTE;
    CEIL5_OUT : BYTE;
  END_VAR

  CEIL5_OUT := BYTE_TO_GRAY(LocalVar0);
END_PROGRAM

CONFIGURATION Config0

  RESOURCE Res0 ON PLC
    TASK task0(INTERVAL := T#20ms,PRIORITY := 0);
    PROGRAM instance0 WITH task0 : program0;
  END_RESOURCE
END_CONFIGURATION

(* ---- BYTE_TO_RANGE.ST ---- *)
FUNCTION _BYTE_TO_REAL:REAL
	VAR_INPUT
		IN :	BYTE;
	END_VAR

	_BYTE_TO_REAL := USINT_TO_REAL(BYTE_TO_USINT(IN));
END_FUNCTION

FUNCTION BYTE_TO_RANGE:REAL
	VAR_INPUT
		X :	BYTE;
		LOW :	REAL;
		HIGH :	REAL;
	END_VAR

	Byte_to_Range := (high - low) * _BYTE_TO_REAL(X) / 255.0 + low;
END_FUNCTION

PROGRAM program0
  VAR
    LocalVar0 : BYTE;
    LocalVar1 : REAL;
	LocalVar2 : REAL;
    CEIL5_OUT : REAL;
  END_VAR

  CEIL5_OUT := BYTE_TO_RANGE(LocalVar0, LocalVar1, LocalVar2);
END_PROGRAM

CONFIGURATION Config0

  RESOURCE Res0 ON PLC
    TASK task0(INTERVAL := T#20ms,PRIORITY := 0);
    PROGRAM instance0 WITH task0 : program0;
  END_RESOURCE
END_CONFIGURATION

(* ---- BYTE_TO_TIME.ST ---- *)
FUNCTION _BYTE_TO_INT:INT
	VAR_INPUT
		IN :	BYTE;
	END_VAR

	_BYTE_TO_INT := USINT_TO_INT(BYTE_TO_USINT(IN));
END_FUNCTION

FUNCTION BYTE_TO_TIME2:TIME
	VAR_INPUT
		IN :	BYTE;
	END_VAR

	BYTE_TO_TIME2 := INT_TO_TIME(_BYTE_TO_INT(IN));
END_FUNCTION

PROGRAM program0
  VAR
    LocalVar0 : BYTE;
    CEIL5_OUT : TIME;
  END_VAR

  CEIL5_OUT := BYTE_TO_TIME2(LocalVar0);
END_PROGRAM

CONFIGURATION Config0

  RESOURCE Res0 ON PLC
    TASK task0(INTERVAL := T#20ms,PRIORITY := 0);
    PROGRAM instance0 WITH task0 : program0;
  END_RESOURCE
END_CONFIGURATION

(* ---- C_TO_F.ST ---- *)
FUNCTION C_TO_F:REAL
	VAR_INPUT
		CELSIUS :	REAL;
	END_VAR

	C_TO_F := celsius * 1.8 + 32.0;
END_FUNCTION

PROGRAM program0
  VAR
    LocalVar0 : REAL;
    CEIL5_OUT : REAL;
  END_VAR

  CEIL5_OUT := C_TO_F(LocalVar0);
END_PROGRAM

CONFIGURATION Config0

  RESOURCE Res0 ON PLC
    TASK task0(INTERVAL := T#20ms,PRIORITY := 0);
    PROGRAM instance0 WITH task0 : program0;
  END_RESOURCE
END_CONFIGURATION

(* ---- C_TO_K.ST ---- *)
FUNCTION C_TO_K:REAL
	VAR_INPUT
		CELSIUS :	REAL;
	END_VAR

	C_to_K := Celsius - 273.15;
END_FUNCTION

PROGRAM program0
  VAR
    LocalVar0 : REAL;
    CEIL5_OUT : REAL;
  END_VAR

  CEIL5_OUT := C_TO_K(LocalVar0);
END_PROGRAM

CONFIGURATION Config0

  RESOURCE Res0 ON PLC
    TASK task0(INTERVAL := T#20ms,PRIORITY := 0);
    PROGRAM instance0 WITH task0 : program0;
  END_RESOURCE
END_CONFIGURATION

(* ---- CAUCHY.ST ---- *)
FUNCTION CAUCHY:REAL
	VAR_INPUT
		X :	REAL;
		T :	REAL;
		U :	REAL;
	END_VAR

	VAR
		tmp :	REAL;
	END_VAR

	tmp := x - t;
	CAUCHY := 0.318309886183791 * U / (U*U + tmp*tmp);
END_FUNCTION

PROGRAM program0
  VAR
    LocalVar0 : REAL;
    LocalVar1 : REAL;
	LocalVar2 : REAL;
    CEIL5_OUT : REAL;
  END_VAR

  CEIL5_OUT := CAUCHY(LocalVar0, LocalVar1, LocalVar2);
END_PROGRAM

CONFIGURATION Config0

  RESOURCE Res0 ON PLC
    TASK task0(INTERVAL := T#20ms,PRIORITY := 0);
    PROGRAM instance0 WITH task0 : program0;
  END_RESOURCE
END_CONFIGURATION

(* ---- CAUCHYCD.ST ---- *)
FUNCTION CAUCHYCD:REAL
	VAR_INPUT
		X :	REAL;
		T :	REAL;
		U :	REAL;
	END_VAR

	CAUCHYCD := 0.5 + 0.318309886183791 * ATAN((X - T) / U);
END_FUNCTION

PROGRAM program0
  VAR
    LocalVar0 : REAL;
	LocalVar1 : REAL;
	LocalVar2 : REAL;
	LocalOUT  : REAL;
  END_VAR
	LocalOUT := CAUCHYCD(LocalVar0, LocalVar1, LocalVar2);
END_PROGRAM

CONFIGURATION Config0
  RESOURCE Res0 ON PLC
    TASK task0(INTERVAL := T#20ms,PRIORITY := 0);
    PROGRAM instance0 WITH task0 : program0;
  END_RESOURCE
END_CONFIGURATION

(* ---- CEIL.ST ---- *)
FUNCTION CEIL:INT

	VAR_INPUT
		X :	REAL;
	END_VAR

	CEIL := REAL_TO_INT(x);
	IF INT_TO_REAL(CEIL) < X THEN
			CEIL := CEIL + 1;
	END_IF;

END_FUNCTION

PROGRAM program0
  VAR
    LocalVar0 : REAL;
    CEIL5_OUT : INT;
  END_VAR

  CEIL5_OUT := CEIL(LocalVar0);
END_PROGRAM

CONFIGURATION Config0

  RESOURCE Res0 ON PLC
    TASK task0(INTERVAL := T#20ms,PRIORITY := 0);
    PROGRAM instance0 WITH task0 : program0;
  END_RESOURCE
END_CONFIGURATION
